# B&R Automation Studio project TD52 (part 55)

### module_EmissionSCR.var - SCR variables
```iecst
VAR
	bAMM_2446 : BOOL := FALSE; (*Warning - SCR BUS communication interrupted [W2446]*) (*V04.05.00.00*)
	bAMM_2447 : BOOL := FALSE; (*Warning - SCR Measuring signal failure urea pressure before dosing [W2447]*) (*V04.05.00.00*)
	bAMM_2448 : BOOL := FALSE; (*Warning - SCR Urea pressure before dosing minimum [W2448]*) (*V04.05.00.00*)
	bAMM_2449 : BOOL := FALSE; (*Warning - SCR Urea pressure before dosing maximum [W2449]*) (*V04.05.00.00*)
	bAMM_2451 : BOOL := FALSE; (*Warning - SCR Urea dosing valve - error [W2451]*) (*V04.05.00.00*)
	bAMM_2452 : BOOL := FALSE; (*Warning - SCR Measuring signal failure urea flow rate after dosing [W2452]*) (*V04.05.00.00*)
	bAMM_2453 : BOOL := FALSE; (*Warning - SCR Urea flow rate - valve characteristic deviating maximum [W2453]*) (*V04.05.00.00*)
	bAMM_2454 : BOOL := FALSE; (*Warning - SCR Compressed air supply pressure urea injection maximum [W2454]*) (*V04.05.00.00*)
	bAMM_2455_CO : BOOL := FALSE; (*Warning - SCR CO Deviation to continous emission monitoring system maximum [W2455]*) (*V04.05.01.00*)
	bAMM_2455_NOx : BOOL := FALSE; (*Warning - SCR NOx Deviation to continous emission monitoring system maximum [W2455]*) (*V04.05.01.00*)
	bAMM_2455_NOxS : BOOL := FALSE; (*Warning - SCR Deviation NOx Sensor to continous emission monitoring system maximum [W2455]*) (*V04.05.01.00*)
	bAMM_2456 : BOOL := FALSE; (*Warning - SCR Emission measurement line 1 - O2 maximum [W2456]*) (*V04.05.00.00*)
	bAMM_2457 : BOOL := FALSE; (*Warning - SCR Measuring signal failure emission measurement line 1 - O2 sensor [W2457]*) (*V04.05.00.00*)
	bAMM_2458 : BOOL := FALSE; (*Warning - SCR Measuring signal failure emission measurement line 2 - NO2 sensor [W2458]*) (*V04.05.00.00*)
	bAMM_2464 : BOOL := FALSE; (*Warning - SCR Urea dosing unit (external) - error [W2464]*) (*V04.05.00.00*)
	bAMM_2697 : BOOL := FALSE; (*Warning - SCR Urea dosing unit - maintenance needed  [W2697]*) (*V04.05.00.00*)
	bAMM_2766 : BOOL := FALSE; (*Warning - Catalyst temperature minimum [W2766]*) (*V04.11.00.00*)
	bAMM_2769 : BOOL := FALSE; (*Warning - SCR Emission measurement air line - moisture maximum [W2769]*) (*V04.14.00.00*)
	bAMM_3379 : BOOL := FALSE; (*Trip - SCR Exhaust temperatures CAT maximum  [A3379]*) (*V04.05.00.00*)
	bAMM_3383 : BOOL := FALSE; (*Trip - SCR Measuring signal failure exhaust temperatures CAT  [A3383]*) (*V04.05.00.00*)
	bAMM_3451 : BOOL := FALSE; (*Warning - SCR Power supply to the valves interrupted [W3451]*) (*V04.05.00.00*)
	bAMM_3452 : BOOL := FALSE; (*Warning - SCR Measuring signal failure urea pressure after dosing [W3452]*) (*V04.05.00.00*)
	bAMM_3453 : BOOL := FALSE; (*Warning - SCR Urea pressure after dosing maximum [W3453]*) (*V04.05.00.00*)
	bAMM_3454 : BOOL := FALSE; (*Warning - SCR Urea pressure after dosing minimum [W3454]*) (*V04.05.00.00*)
	bAMM_3455 : BOOL := FALSE; (*Warning - SCR Urea flow rate after dosing maximum [W3455]*) (*V04.05.00.00*)
	bAMM_3456 : BOOL := FALSE; (*Warning - SCR Urea dosing pump - error [W3456]*) (*V04.05.00.00*)
	bAMM_3457 : BOOL := FALSE; (*Warning - SCR Urea-air valve blocked [W3457]*) (*V04.05.00.00*)
	bAMM_3459 : BOOL := FALSE; (*Warning - SCR Urea tank level minimum - dosing deactivated [W3459]*) (*V04.05.00.00*)
	bAMM_3460 : BOOL := FALSE; (*Warning - SCR Urea supply pump not operating [W3460]*) (*V04.05.00.00*)
	bAMM_3461 : BOOL := FALSE; (*Warning - SCR Measuring signal failure compressed air supply pressure urea injection [W3461]*) (*V04.05.00.00*)
	bAMM_3462 : BOOL := FALSE; (*Warning - SCR Compressed air supply pressure urea injection minimum [W3462]*) (*V04.05.00.00*)
	bAMM_3463 : BOOL := FALSE; (*Warning - SCR Compressed air valve urea injection power supply interrupted [W3463]*) (*V04.05.00.00*)
	bAMM_3464 : BOOL := FALSE; (*Warning - SCR Measuring signal failure exhaust pressure CAT inlet [W3464]*) (*V04.05.00.00*)
	bAMM_3465 : BOOL := FALSE; (*Warning - SCR Measuring signal failure exhaust pressure CAT outlet [W3465]*) (*V04.05.00.00*)
	bAMM_3466 : BOOL := FALSE; (*Warning - SCR Measuring signal failure exhaust temperature CAT inlet [W3466]*) (*V04.05.00.00*)
	bAMM_3467 : BOOL := FALSE; (*Warning - SCR Measuring signal failure exhaust temperature CAT outlet [W3467]*) (*V04.05.00.00*)
	bAMM_3469 : BOOL := FALSE; (*Warning - SCR Exhaust differential pressure CAT maximum [W3469]*) (*V04.05.00.00*)
	bAMM_3470 : BOOL := FALSE; (*Warning - SCR Emission measurement sample gas cooler - error [W3470]*) (*V04.05.00.00*)
	bAMM_3471 : BOOL := FALSE; (*Warning - SCR Emission measurement line 1 - sample gas pump not ready [W3471]*) (*V04.05.00.00*)
	bAMM_3472 : BOOL := FALSE; (*Warning - SCR Emission measurement line 2 - sample gas pump not ready [W3472]*) (*V04.05.00.00*)
	bAMM_3473 : BOOL := FALSE; (*Warning - SCR Emission measurement line 1 - moisture maximum [W3473]*) (*V04.05.00.00*)
	bAMM_3474 : BOOL := FALSE; (*Warning - SCR Emission measurement line 2 - moisture maximum [W3474]*) (*V04.05.00.00*)
	bAMM_3475 : BOOL := FALSE; (*Warning - SCR Emission measurement line 1 - flow rate minimum [W3475]*) (*V04.05.00.00*)
	bAMM_3476 : BOOL := FALSE; (*Warning - SCR Emission measurement line 2 - flow rate minimum [W3476]*) (*V04.05.00.00*)
	bAMM_3477 : BOOL := FALSE; (*Warning - SCR Measuring signal failure emission measurement line 2 - NO sensor [W3477]*) (*V04.05.00.00*)
	bAMM_3478 : BOOL := FALSE; (*Warning - SCR Measuring signal failure emission measurement line 1 - NO sensor [W3478]*) (*V04.05.00.00*)
	bAMM_3479 : BOOL := FALSE; (*Warning - SCR Measuring signal failure emission measurement line 1 - NO2 sensor [W3479]*) (*V04.05.00.00*)
	bAMM_3480 : BOOL := FALSE; (*Warning - SCR NH3 slip detection deactivated  [W3480]*) (*V04.05.00.00*)
	bAMM_3481 : BOOL := FALSE; (*Warning - SCR Measuring signal failure emission measurement line 1 - CO sensor [W3481]*) (*V04.05.00.00*)
	bAMM_3486 : BOOL := FALSE; (*Warning - SCR Urea flow rate after dosing minimum [W3486]*) (*V04.05.00.00*)
	bAMM_3487 : BOOL := FALSE; (*Warning - SCR Exhaust temperature CAT inlet maximum [W3487]*) (*V04.05.00.00*)
	bAMM_3488 : BOOL := FALSE; (*Warning - SCR Exhaust temperature CAT outlet maximum [W3488]*) (*V04.05.00.00*)
	bAMM_9212 : BOOL := FALSE; (*Warning - SCR Air compressor - maintenance needed [W9212]*) (*V04.05.00.00*)
	bAMM_9277 : BOOL := FALSE; (*Warning - SCR Urea dosing stopped - error [W9277]*) (*V04.07.00.00*)
	bAMM_9379 : BOOL := FALSE; (*Warning - SCR Measuring signal failure urea tank level [W9379]*) (*V04.13.00.00*)
	bAMM_9380 : BOOL := FALSE; (*Warning - SCR Urea flow dosing error [W9380]*) (*V04.13.00.00*)
	bEMLine1_Exist : BOOL := FALSE; (*SCR Emission measurement line 1 - exist*) (*V04.13.00.00*)
	bEMLine2_Exist : BOOL := FALSE; (*SCR Emission measurement line 2 - exist*) (*V04.13.00.00*)
	bErr_SCR_BUS : BOOL := FALSE; (*SCR: Bus communication not ok*) (*V04.05.00.00*)
	bOpM_2878 : BOOL := FALSE; (*Operational message - SCR Urea dosing activated  [B2878]*) (*V04.05.00.00*)
	bOpM_2879 : BOOL := FALSE; (*Operational message - SCR Urea dosing deactivated  [B2879]*) (*V04.05.00.00*)
	bOpM_2884 : BOOL := FALSE; (*Operational message - SCR Manual mode on [B2884]*) (*V04.05.00.00*)
	bOpM_2885 : BOOL := FALSE; (*Operational message - SCR Manual mode off [B2885]*) (*V04.05.00.00*)
	bOpM_2923 : BOOL := FALSE; (*Operational message - SCR NH3 slip detection started  [B2923]*) (*V04.05.00.00*)
	bOpM_2924 : BOOL := FALSE; (*Operational message - SCR NH3 slip detection completed  [B2924]*) (*V04.05.00.00*)
	bOpM_9077 : BOOL := FALSE; (*Operational message - SCR NH3 slip detection interrupted  [B9077]*) (*V04.13.00.00*)
	bOpM_9079 : BOOL := FALSE; (*Operational message - SCR Urea dosing - dosing conditions reached [B9079]*) (*V04.13.00.00*)
	bOpM_9080 : BOOL := FALSE; (*Operational message - SCR Urea dosing - dosing conditions ended [B9080]*) (*V04.13.00.00*)
	bOpM_9081 : BOOL := FALSE; (*Operational message - SCR Urea dosing - requested [B9081]*) (*V04.13.00.00*)
	bOpM_9082 : BOOL := FALSE; (*Operational message - SCR Urea dosing - unrequested [B9082]*) (*V04.13.00.00*)
	bRelMon_Lev_UreaTank : BOOL := FALSE; (*release monitoring - urea tank level measuring *) (*V04.13.00.00*)
	bRelMon_T_CatIn : BOOL := FALSE; (*release monitoring - temperature before catalyst*) (*V04.05.00.00*)
	bRelMon_T_CatOut : BOOL := FALSE; (*release monitoring - temperature after catalyst*) (*V04.05.00.00*)
	bRel_Dosing : BOOL := FALSE; (*release dosing*) (*V04.05.00.00*)
	bRel_SCR_UDC : BOOL := FALSE; (*SCR Release urea dosing controller (UDC)*) (*V04.05.00.00*)
	bSCR_DosingLimReached : BOOL := FALSE; (*SCR Limits for dosing release reached*) (*V04.07.00.00*)
END_VAR
VAR CONSTANT
	MODBUS_RTU_MASTER_MAX_ARRAY : UINT := 400; (*Max data (INT) to send/receive *) (*V04.05.00.00*)
END_VAR
VAR
	tInternFlow_SCR_UreaDosingOut : HALioAi_Type; (*SCR Urea flow rate after dosing unit [l/h] (INTERNAL)*) (*V04.05.00.00*)
	tInternPr_SCR_ComprAirSupply : HALioAi_Type; (*SCR Compressed air supply pressure urea injection [bar] (INTERNAL)*) (*V04.05.00.00*)
	tInternPr_SCR_UreaDosingIn : HALioAi_Type; (*SCR Urea pressure before dosing unit [bar] (INTERNAL)*) (*V04.05.00.00*)
	tInternPr_SCR_UreaDosingOut : HALioAi_Type; (*SCR Urea pressure after dosing unit [bar] (INTERNAL)*) (*V04.05.00.00*)
	tInternSCR_InjectValve_Air : HALioDi_Type; (*SCR Urea/Air injection valve - air opened (INTERNAL)*) (*V04.05.00.00*)
	tInternSCR_InjectValve_Urea : HALioDi_Type; (*SCR Urea/Air injection valve - urea opened (INTERNAL)*) (*V04.05.00.00*)
	xTON_bRel_SCR_UDC_5m : TON := (0); (*FuB*)
	xUDC : fUDC := (0); (*FuB*) (*V04.05.00.00*)
END_VAR
```

### Program Logical/Emission/GeneralEM (IEC, version 4.14.0) - general functions

#### GeneralEMCyclic.st
```iecst
(*******************************************************************************
GeneralEM		general functions

This code is confidential and proprietary to the INNIO Company.
It may not be used in any form, or reproduced in any manner,
without the express written permission of the INNIO Company.
Copyright, INNIO Company, 2019

Customized modifications: -
------------------------

History:
-------
V04.05.00.00	22.05.2017	Tinello		new
V04.05.06.00	16.07.2018	Tinello 	Bugfix start speed, bu
V04.07.00.00	11.04.2019	Tinello 	engine motortype included
V04.14.00.00	18.11.2024	Farre		added NOx sensor selection: standard or Low (2023-183)

Instructions for use:
--------------------
Outstandings:
------------
*******************************************************************************)
PROGRAM _CYCLIC

	(* Release Module if ParaSetupOk = TRUE *)
	xTON_ParaSetupOk(IN		:= IN_EM.tPB2MM.bParaSetupOk, PT:= T#10s);
	bRelModul_ParaSetupOk	:= xTON_ParaSetupOk.Q;

	(* operation mode *)
	xOpMode.in	:=	IN_EM.iSt_OpMode;
	xOpMode();

	(* Operation mode selector switch *) 	(* 1= manual; 2= auto; 3= test mode *)
	xTOF_OMSS_MAT(IN	:= (IN_EM.iIdx_OMSS = 1) OR (IN_EM.iIdx_OMSS = 2) OR (IN_EM.iIdx_OMSS = 3), PT := T#10m);
	bOMSS_MAT			:= xTOF_OMSS_MAT.IN;
	bOMSS_MAT_TOF_10m	:= xTOF_OMSS_MAT.Q;

	(* engine start speed reached *)
	xGR_MAXR_StartSpd(In:= IN_EM.rN_EngAct,   Gw := Para.rN_EngStart_LimHi, Hy := Para.rN_EngStart_HyHi);
	xTOF_StartSpd(IN 	:= xGR_MAXR_StartSpd.Q AND bRelModul_ParaSetupOk, 	PT := T#10s);
	xTON_StartSpd_5m(IN := xGR_MAXR_StartSpd.Q AND bRelModul_ParaSetupOk, 	PT := T#5m);

	bStartSpd			:= xTOF_StartSpd.Q;
	bStartSpd_5m		:= xTON_StartSpd_5m.Q;

	(* Engine motortype *)
	xEngType.Motortype 	:= INT_TO_UINT(Para.iEng_Motortype);
	xEngType();

	(* Type of device installed after catalyst *)
	bNOxS_CatOut_Std 	:= Para.iNOxS_CatOut_Device_Type = 0;				(* 0: Standard NOx sensor *)
	bNOxS_CatOut_Low 	:= Para.iNOxS_CatOut_Device_Type = 1;				(* 1: Low NOx sensor *)

END_PROGRAM
```

#### GeneralEM.var
```iecst
VAR
	xGR_MAXR_StartSpd : GR_MAXR := (0); (*Engine start speed passed*)
	xTOF_OMSS_MAT : TOF := (0); (*FuB*)
	xTOF_StartSpd : TOF := (0); (*FuB*)
	xTON_ParaSetupOk : TON := (0); (*FuB*)
	xTON_StartSpd_5m : TON := (0); (*FuB*)
END_VAR
```

### Program Logical/Emission/DefaultEM (IEC, version 4.07.0) - Settings default values

#### DefaultEMCyclic.st
```iecst
(*******************************************************************************
DefaultEM		value set

This code is confidential and proprietary to the INNIO Company.
It may not be used in any form, or reproduced in any manner,
without the express written permission of the INNIO Company.
Copyright, INNIO Company, 2019

Customized modifications: -
------------------------

History:
-------
V4.05.0	05.04.2017	Tinello		new
V4.07.0	23.01.2019	Tinello		add Customer DI's

Instructions for use:
--------------------
Outstandings:
------------
*******************************************************************************)
PROGRAM _CYCLIC

	(* SCR *)
	IN_EM.tFS_SCR_EMLine1_Lo.Di				:= IN_EM.tFS_SCR_EMLine1_Lo.Di				OR NOT IN_EM.tFS_SCR_EMLine1_Lo.GoodQual;
	IN_EM.tFS_SCR_EMLine2_Lo.Di				:= IN_EM.tFS_SCR_EMLine2_Lo.Di				OR NOT IN_EM.tFS_SCR_EMLine2_Lo.GoodQual;
	IN_EM.tLev_SCR_UreaDosingCabinet_Hi.Di	:= IN_EM.tLev_SCR_UreaDosingCabinet_Hi.Di	OR NOT IN_EM.tLev_SCR_UreaDosingCabinet_Hi.GoodQual;
	IN_EM.tLev_SCR_UreaTank_Lo.Di			:= IN_EM.tLev_SCR_UreaTank_Lo.Di			OR NOT IN_EM.tLev_SCR_UreaTank_Lo.GoodQual;
	IN_EM.tSCR_AirCompressor_Rdy.Di			:= IN_EM.tSCR_AirCompressor_Rdy.Di			OR NOT IN_EM.tSCR_AirCompressor_Rdy.GoodQual;
	IN_EM.tSCR_ComprAirValve_Rdy.Di			:= IN_EM.tSCR_ComprAirValve_Rdy.Di			OR NOT IN_EM.tSCR_ComprAirValve_Rdy.GoodQual;
	IN_EM.tSCR_EMCooler_Rdy.Di				:= IN_EM.tSCR_EMCooler_Rdy.Di				OR NOT IN_EM.tSCR_EMCooler_Rdy.GoodQual;
	IN_EM.tSCR_EMPump1_Rdy.Di				:= IN_EM.tSCR_EMPump1_Rdy.Di				OR NOT IN_EM.tSCR_EMPump1_Rdy.GoodQual;
	IN_EM.tSCR_EMPump2_Rdy.Di				:= IN_EM.tSCR_EMPump2_Rdy.Di				OR NOT IN_EM.tSCR_EMPump2_Rdy.GoodQual;
	IN_EM.tSCR_UreaDosingPump_Rdy.Di		:= IN_EM.tSCR_UreaDosingPump_Rdy.Di			OR NOT IN_EM.tSCR_UreaDosingPump_Rdy.GoodQual;
	IN_EM.tSCR_UreaDosingPump2_Rdy.Di		:= IN_EM.tSCR_UreaDosingPump2_Rdy.Di		OR NOT IN_EM.tSCR_UreaDosingPump2_Rdy.GoodQual;
	IN_EM.tSCR_UreaSupplyPump_Op.Di			:= IN_EM.tSCR_UreaSupplyPump_Op.Di			OR NOT IN_EM.tSCR_UreaSupplyPump_Op.GoodQual;
	IN_EM.tSCR_ValvePowerSupply_Ok.Di		:= IN_EM.tSCR_ValvePowerSupply_Ok.Di		OR NOT IN_EM.tSCR_ValvePowerSupply_Ok.GoodQual;
	IN_EM.tSCR_InjectValve_Opened.Di		:= IN_EM.tSCR_InjectValve_Opened.Di			OR NOT IN_EM.tSCR_InjectValve_Opened.GoodQual;
	IN_EM.tSCR_Catalyst_Rdy.Di				:= IN_EM.tSCR_Catalyst_Rdy.Di				OR NOT IN_EM.tSCR_Catalyst_Rdy.GoodQual;
	IN_EM.tT_SCR_Cat_HiHi.Di				:= IN_EM.tT_SCR_Cat_HiHi.Di					OR NOT IN_EM.tT_SCR_Cat_HiHi.GoodQual;
END_PROGRAM
```

### Program Logical/Emission/EmissionMon (IEC, version 4.11.0) - + Emission Monitoring 

- EmissionMon.st (not readable text: treated as protected, skipped)

#### EmissionMon.var - Local variables
```iecst
VAR
	bAMM_NOx_Em_AvgDaily_Hi_Ack : BOOL := FALSE; (*NOx emissions - daily average high warning - acknowledgeable*)
	bNewDay : BOOL := FALSE; (*day changed*)
	bNOxValue_Valid : BOOL := FALSE; (*Valid NOx value available*)
	bNOx_Em_EngOut_mg_LoadSet_Save : BOOL := FALSE; (*SAVE Parameter value: NOx emissions at the engine outlet - Load dependent setpoint enable*)
	bP_Act_Min_reached : BOOL := FALSE; (*Minimal power reached*)
	bRelMon_NOx_Em_Avg : BOOL := FALSE; (*Release monitoring of NOx average*)
	i : INT := 0; (*auxiliary variable*)
	iCnt_Em_AvgShort : UINT := 0; (*counter - for average calculation - NOx and CO short-term*)
	iCnt_MonLim_Exc : UINT; (*counter for emission tolerance exceedance [s]*)
	rCO_Em_AvgShort_Sum_mg : REAL := 0; (*Sum for average calculation - CO short-term [mg/Nm3]*)
	rCO_Em_Avg_mg : ARRAY[0..1799] OF REAL := [1800(0)]; (*Up to 1800 values (300min) for average calculation of CO [mg/Nm3]*)
	rCO_Em_CatOut_mg : REAL := 0; (*Actual CO value at catalyst outlet [mg/Nm3]*)
	rNO2_Em_CatOut_mg : REAL := 0; (*Actual NO2 value at catalyst outlet [mg/Nm3]*)
	rNOx_Em_AvgShort_Sum_mg : REAL := 0; (*Sum for average calculation - NOx short-term [mg/Nm3]*)
	rNOx_Em_Avg_mg : ARRAY[0..1799] OF REAL := [1800(0)]; (*Up to 1800 values (300min) for average calculation of NOx [mg/Nm3]*)
	rNOx_Em_EngOut_mg_Set_Int : REAL := 0; (*INTERNAL: NOx emissions at engine outlet - setpoint [mg/Nm3]*)
	rNOx_NOxS_CatOut_mg : REAL := 0; (*Actual NOx value at catalyst outlet from NOx sensor [mg/Nm3]*)
	rNO_Em_CatOut_mg : REAL := 0; (*Actual NO value at catalyst outlet [mg/Nm3]*)
	rP_Set_Min_NormHy : REAL := 0; (*Minimal power setpoint related to rP_nom -  hysteresis*)
	tRealTime : rtctime_typ; (*actual time of controller*)
	tRefPoint_NOx_mg_Set : ARRAY[0..3] OF lcrCurveByPoints_TabEntry_type; (*kW/NOx Points for interpolation of NOx emissions at engine outlet - setpoint [mg/Nm3]*)
	xDTGetTime_RPS : DTGetTime; (*getting time of the controller*)
	xFILTER_R_NOx_mg_Set : FILTER_R := (0); (*FuB*)
	xFILTER_R_O2_EngOut_Avg : FILTER_R := (0); (*FuB*)
	xLCRCurveByPoints_NOx_mg_Set : LCRCurveByPoints := (0); (*FuB*)
	xLCRMovAvgFlt_CO_short : LCRMovAvgFlt := (0); (*FuB*)
	xLCRMovAvgFlt_NOx_daily : LCRMovAvgFlt := (0); (*FuB*)
	xLCRMovAvgFlt_NOx_dailyT : LCRMovAvgFlt := (0); (*FuB*)
	xLCRMovAvgFlt_NOx_short : LCRMovAvgFlt := (0); (*FuB*)
	xTON_10sec_Tick : TON := (0); (*FuB*)
	xTON_CO_Hi_1 : TON := (0); (*FuB*)
	xTON_DosExt_3m : TON := (0); (*FuB*)
	xTON_EngineSteadyState : TON := (0); (*FuB*)
	xTON_GasAnalys_Done : TON := (0); (*FuB*)
	xTON_NOx_Hi_1 : TON := (0); (*FuB*)
	xTON_NOx_Hi_2 : TON := (0); (*FuB*)
	xTON_P_Act_MinHy : TON := (0); (*FuB*)
	xTON_P_Min_02m : TON := (0); (*FuB*)
	xTON_P_Min_20m : TON := (0); (*FuB*)
	xTON_SecondTick : TON := (0); (*FuB*)
	xTON_StartupDone : TON := (0); (*FuB*)
	xTP_30s : TP; (*FuB*)
END_VAR
```

### Program Logical/Emission/NOxSensor (IEC, version 4.14.0) - + Read Nox Data

- NOxSensor.st (not readable text: treated as protected, skipped)

#### NOxSensor.var - Local variables
```iecst
VAR
	bAMM_NOxS_CANrd_CatOut : BOOL := FALSE; (*Warning: No connection to the sensor - NOx sensor CAT out*) (*OldName: newPV; Cycle: 5*)
	bAMM_NOxS_CANrd_EngOut : BOOL := FALSE; (*Warning: No connection to the sensor - NOx sensor engine out*) (*OldName: newPV; Cycle: 5*)
	bAMM_NOxS_CANrd_EngOut_A : BOOL := FALSE; (*Warning: No connection to the sensor - NOx sensor engine out bank A*) (*OldName: newPV; Cycle: 5*)
	bAMM_NOxS_CANrd_EngOut_B : BOOL := FALSE; (*Warning: No connection to the sensor - NOx sensor engine out bank B*) (*OldName: newPV; Cycle: 5*)
	bDewpoint_NOxS1_IF1 : BOOL := FALSE; (*NOx sensors 1 at CAN interface 1 - Dewpoint reached/sensor started*) (*OldName: newPV; Cycle: 5*)
	bDewpoint_NOxS2_IF1 : BOOL := FALSE; (*NOx sensors 2 at CAN interface 1 - Dewpoint reached/sensor started*) (*OldName: newPV; Cycle: 5*)
	bDewpoint_NOxS2_IF2 : BOOL := FALSE; (*NOx sensors 2 at CAN interface 2 - Dewpoint reached/sensor started*) (*OldName: newPV; Cycle: 5*)
	bDewP_Reached_CatOut : BOOL := FALSE; (*Dew point reached - CAT out*) (*OldName: newPV; Cycle: 5*)
	bDewP_Reached_EngOut : BOOL := FALSE; (*Dew point reached - engine out*) (*OldName: newPV; Cycle: 5*)
	bNOxS_CatOut_Diag_Req : BOOL := FALSE; (*NOx sensor - CAT out- self diagnosis request*) (*OldName: newPV; Cycle: 5*)
	bNOxS_CatOut_Diag_Active : BOOL := FALSE; (*NOx sensor - CAT out - self diagnosis active*) (*OldName: newPV; Cycle: 5*)
	bNOxS_EngOut_A_Diag_Active : BOOL := FALSE; (*NOx sensor - engine out bank A - self diagnosis active*) (*OldName: newPV; Cycle: 5*)
	bNOxS_EngOut_A_Diag_Req : BOOL := FALSE; (*NOx sensor - engine out bank A - self diagnosis request *) (*OldName: newPV; Cycle: 5*)
	bNOxS_EngOut_B_Diag_Active : BOOL := FALSE; (*NOx sensor - engine out bank B - self diagnosis active*) (*OldName: newPV; Cycle: 5*)
	bNOxS_EngOut_B_Diag_Req : BOOL := FALSE; (*NOx sensor - engine out bank B - self diagnosis request *) (*OldName: newPV; Cycle: 5*)
	bNOxS_EngOut_Diag_Active : BOOL := FALSE; (*NOx sensor - engine out - self diagnosis active*) (*OldName: newPV; Cycle: 5*)
	bNOxS_EngOut_Diag_Req : BOOL := FALSE; (*NOx sensor - engine out - self diagnosis request *) (*OldName: newPV; Cycle: 5*)
	bQueue_NOxS1_IF1_Done : BOOL := FALSE; (*initialisation of CAN queue for NOx sensor 1 (interface1) is done*) (*OldName: newPV; Cycle: 5*)
	bQueue_NOxS2_IF1_Done : BOOL := FALSE; (*initialisation of CAN queue for NOx sensor 2 (interface1) is done*) (*OldName: newPV; Cycle: 5*)
	bQueue_NOxS2_IF2_Done : BOOL := FALSE; (*initialisation of CAN queue for NOx sensor 2 (interface2) is done*) (*OldName: newPV; Cycle: 5*)
	bRelMon_O2_NOxS_CatOut : BOOL := FALSE; (*Release monitoring NOx sensor at CAT outlet - O2 value*) (*OldName: newPV; Cycle: 5*)
	bRelMon_O2_NOxS_EngOut : BOOL := FALSE; (*Release monitoring NOx sensor at engine outlet - O2 value*) (*OldName: newPV; Cycle: 5*)
	bRelMon_O2_NOxS_EngOut_A : BOOL := FALSE; (*Release monitoring NOx sensor at engine outlet bank A - O2 value*) (*OldName: newPV; Cycle: 5*)
	bRelMon_O2_NOxS_EngOut_B : BOOL := FALSE; (*Release monitoring NOx sensor at engine outlet bank B - O2 value*) (*OldName: newPV; Cycle: 5*)
	bReq_NOxS1_IF1_CF : BOOL := FALSE; (*request correction factor for NOx sensor 1 (interface1)*) (*OldName: newPV; Cycle: 5*)
	bReq_NOxS1_IF1_DiagRes : BOOL := FALSE; (*request self diagnosis result value for NOx sensor 1 (interface1)*) (*OldName: newPV; Cycle: 5*)
	bReq_NOxS1_IF1_OpH : BOOL := FALSE; (*request operating hours for NOx sensor 1 (interface1)*) (*OldName: newPV; Cycle: 5*)
	bReq_NOxS2_IF1_CF : BOOL := FALSE; (*request correction factor for NOx sensor 2 (interface1)*) (*OldName: newPV; Cycle: 5*)
	bReq_NOxS2_IF1_DiagRes : BOOL := FALSE; (*request self diagnosis result value for NOx sensor 2 (interface1)*) (*OldName: newPV; Cycle: 5*)
	bReq_NOxS2_IF1_OpH : BOOL := FALSE; (*request operating hours for NOx sensor 2 (interface1)*) (*OldName: newPV; Cycle: 5*)
	bReq_NOxS2_IF2_CF : BOOL := FALSE; (*request correction factor for NOx sensor 2 (interface2)*) (*OldName: newPV; Cycle: 5*)
	bReq_NOxS2_IF2_DiagRes : BOOL := FALSE; (*request self diagnosis result value for NOx sensor 2 (interface2)*) (*OldName: newPV; Cycle: 5*)
	bReq_NOxS2_IF2_OpH : BOOL := FALSE; (*request operating hours for NOx sensor 2 (interface2)*) (*OldName: newPV; Cycle: 5*)
	bStart_NOxS_CatOut : BOOL := FALSE; (*NOx sensor - CAT out - start command*) (*OldName: newPV; Cycle: 5*)
	bStart_NOxS_EngOut : BOOL := FALSE; (*NOx sensor - engine out - start command*) (*OldName: newPV; Cycle: 5*)
	DATA_NOxS_R : ARRAY[0..7] OF USINT; (*read data from NOx sensor*) (*OldName: newPV; Cycle: 5*)
	DATA_NOxS_W : ARRAY[0..2] OF USINT; (*request data from NOx sensor*) (*OldName: newPV; Cycle: 5*)
	i : UINT := 0; (*auxiliaries variable*) (*OldName: newPV; Cycle: 5*)
	iAlternate_Req : USINT := 0; (*Alternate request*) (*OldName: newPV; Cycle: 5*)
	iCANqueue_NOxS_size : UINT := 0; (*CANqueue size*) (*OldName: newPV; Cycle: 5*)
	iCANwrite_NOxS_Diag_IF1 : ARRAY[0..7] OF USINT; (*Message for NOx sensors CAN interface 1 - self diagnosis*) (*OldName: newPV; Cycle: 5*)
	iCANwrite_NOxS_Diag_IF2 : ARRAY[0..7] OF USINT; (*Message for NOx sensors CAN interface 2 - self diagnosis*) (*OldName: newPV; Cycle: 5*)
	iCANwrite_NOxS_IF1 : ARRAY[0..7] OF USINT; (*Message for NOx sensors CAN interface 1*) (*OldName: newPV; Cycle: 5*)
	iCANwrite_NOxS_IF1_Old : USINT := 0; (*Message for NOx sensors CAN interface 1 - saved*) (*OldName: newPV; Cycle: 5*)
	iCANwrite_NOxS_IF2 : ARRAY[0..7] OF USINT; (*Message for NOx sensors CAN interface 2*) (*OldName: newPV; Cycle: 5*)
	iCANwrite_NOxS_IF2_Old : USINT := 0; (*Message for NOx sensors CAN interface 2 - saved*) (*OldName: newPV; Cycle: 5*)
	iCAN_NOxS_us_ident : UDINT; (*identifier for CAN read/write*) (*OldName: newPV; Cycle: 5*)
	iCnt_NOxS_CatOut_Diag : USINT := 0; (*Counter - NOx sensor catalyst out - diagnosis counter*) (*OldName: newPV; Cycle: 5*)
	iCnt_NOxS_EngOut_A_Diag : USINT := 0; (*Counter - NOx sensor engine out A - diagnosis counter*) (*OldName: newPV; Cycle: 5*)
	iCnt_NOxS_EngOut_B_Diag : USINT := 0; (*Counter - NOx sensor engine out B - diagnosis counter*) (*OldName: newPV; Cycle: 5*)
	iCnt_NOxS_EngOut_Diag : USINT := 0; (*Counter - NOx sensor engine out - diagnosis counter*) (*OldName: newPV; Cycle: 5*)
	iCnt_NOx_NOxS_CatOut_Err : USINT := 0; (*Counter - NOx sensor catalyst out - error NOx*) (*OldName: newPV; Cycle: 5*)
	iCnt_NOx_NOxS_EngOut_A_Err : USINT := 0; (*Counter - NOx sensor engine out A - error NOx*) (*OldName: newPV; Cycle: 5*)
	iCnt_NOx_NOxS_EngOut_B_Err : USINT := 0; (*Counter - NOx sensor engine out B - error NOx*) (*OldName: newPV; Cycle: 5*)
	iCnt_NOx_NOxS_EngOut_Err : USINT := 0; (*Counter - NOx sensor engine out - error NOx*) (*OldName: newPV; Cycle: 5*)
	iCnt_O2_NOxS_CatOut_Err : USINT := 0; (*Counter - NOx sensor catalyst out - error O2*) (*OldName: newPV; Cycle: 5*)
	iCnt_O2_NOxS_EngOut_A_Err : USINT := 0; (*Counter - NOx sensor engine out A - error O2*) (*OldName: newPV; Cycle: 5*)
	iCnt_O2_NOxS_EngOut_B_Err : USINT := 0; (*Counter - NOx sensor engine out B - error O2*) (*OldName: newPV; Cycle: 5*)
	iCnt_O2_NOxS_EngOut_Err : USINT := 0; (*Counter - NOx sensor engine out - error O2*) (*OldName: newPV; Cycle: 5*)
	iCnt_OpHours_Old : DINT; (*Save operating hours*) (*OldName: newPV; Cycle: 5*)
	iCnt_RequestTrials : ARRAY[0..9] OF USINT; (*Number of request trials*) (*OldName: newPV; Cycle: 5*)
	iCnt_Wait : USINT := 0; (*Cycle counter - wait for CAN message*) (*OldName: newPV; Cycle: 5*)
	iCnt_WaitErrS1_IF1 : USINT := 0; (*Cycle counter - error while waiting for CAN message*) (*OldName: newPV; Cycle: 5*)
	iCnt_WaitErrS2_IF1 : USINT := 0; (*Cycle counter - error while waiting for CAN message*) (*OldName: newPV; Cycle: 5*)
	iCnt_WaitErrS2_IF2 : USINT := 0; (*Cycle counter - error while waiting for CAN message*) (*OldName: newPV; Cycle: 5*)
	iCnt_WaitS1_IF1 : USINT := 0; (*Cycle counter - wait for CAN message*) (*OldName: newPV; Cycle: 5*)
	iCnt_WaitS2_IF1 : USINT := 0; (*Cycle counter - wait for CAN message*) (*OldName: newPV; Cycle: 5*)
	iCnt_WaitS2_IF2 : USINT := 0; (*Cycle counter - wait for CAN message*) (*OldName: newPV; Cycle: 5*)
	iIdx_NOxS_Config_Old : INT := 0; (*Save - PARA: NOx  Sensor configuration*) (*OldName: newPV; Cycle: 5*)
	iNOx_NOxS_CatOut_Wet : UINT := 0; (*NOx sensor catalyst out - assembly high and low byte of NOx*) (*OldName: newPV; Cycle: 5*)
	iNOx_NOxS_EngOut_A_Wet : UINT := 0; (*NOx sensor engine out A - assembly high and low byte of NOx*) (*OldName: newPV; Cycle: 5*)
	iNOx_NOxS_EngOut_B_Wet : UINT := 0; (*NOx sensor engine out B - assembly high and low byte of NOx*) (*OldName: newPV; Cycle: 5*)
	iNOx_NOxS_EngOut_Wet : UINT := 0; (*NOx sensor engine out - assembly high and low byte of NOx*) (*OldName: newPV; Cycle: 5*)
	iO2_NOxS_CatOut_Wet : UINT := 0; (*NOx sensor catalyst out - assembly high and low byte of O2*) (*OldName: newPV; Cycle: 5*)
	iO2_NOxS_EngOut_A_Wet : UINT := 0; (*NOx sensor engine out A - assembly high and low byte of O2*) (*OldName: newPV; Cycle: 5*)
	iO2_NOxS_EngOut_B_Wet : UINT := 0; (*NOx sensor engine out B - assembly high and low byte of O2*) (*OldName: newPV; Cycle: 5*)
	iO2_NOxS_EngOut_Wet : UINT := 0; (*NOx sensor engine out - assembly high and low byte of O2*) (*OldName: newPV; Cycle: 5*)
	iRead_NOxS_CatOut : ARRAY[0..7] OF USINT; (*CAN data - NOx sensor catalyst out*) (*OldName: newPV; Cycle: 5*)
	iRead_NOxS_EngOut : ARRAY[0..7] OF USINT; (*CAN data - NOx sensor engine out*) (*OldName: newPV; Cycle: 5*)
	iRead_NOxS_EngOut_A : ARRAY[0..7] OF USINT; (*CAN data - NOx sensor engine out A*) (*OldName: newPV; Cycle: 5*)
	iRead_NOxS_EngOut_B : ARRAY[0..7] OF USINT; (*CAN data - NOx sensor engine out B*) (*OldName: newPV; Cycle: 5*)
	iSel_NOxS_Request : USINT := 0; (*Selection of CAN request*) (*OldName: newPV; Cycle: 5*)
	iSt_NOxS_CatOut_Diagnosis : USINT := 0; (*NOx sensor catalyst out - status diagnosis feedback*) (*OldName: newPV; Cycle: 5*)
	iSt_NOxS_CatOut_HeaterErr : USINT := 0; (*NOx sensor catalyst out - status heater error*) (*OldName: newPV; Cycle: 5*)
	iSt_NOxS_CatOut_HeaterMode : USINT := 0; (*NOx sensor catalyst out - status heater mode*) (*OldName: newPV; Cycle: 5*)
	iSt_NOxS_CatOut_HeaterTemp : USINT := 0; (*NOx sensor catalyst out - status temperature heater*) (*OldName: newPV; Cycle: 5*)
	iSt_NOxS_CatOut_NOxErr : USINT := 0; (*NOx sensor catalyst out - status NOx error*) (*OldName: newPV; Cycle: 5*)
	iSt_NOxS_CatOut_NOxSignal : USINT := 0; (*NOx sensor catalyst out - status NOx signal*) (*OldName: newPV; Cycle: 5*)
	iSt_NOxS_CatOut_O2Err : USINT := 0; (*NOx sensor catalyst out - status Oxygen error*) (*OldName: newPV; Cycle: 5*)
	iSt_NOxS_CatOut_O2Signal : USINT := 0; (*NOx sensor catalyst out - status Oxygen signal*) (*OldName: newPV; Cycle: 5*)
	iSt_NOxS_CatOut_PowerRange : USINT := 0; (*NOx sensor catalyst out - status power in range*) (*OldName: newPV; Cycle: 5*)
	iSt_NOxS_EngOut_A_Diagnosis : USINT := 0; (*NOx sensor engine out A - status diagnosis feedback*) (*OldName: newPV; Cycle: 5*)
	iSt_NOxS_EngOut_A_HeaterErr : USINT := 0; (*NOx sensor engine out A - status heater error*) (*OldName: newPV; Cycle: 5*)
	iSt_NOxS_EngOut_A_HeaterMode : USINT := 0; (*NOx sensor engine out A - status heater mode*) (*OldName: newPV; Cycle: 5*)
	iSt_NOxS_EngOut_A_HeaterTemp : USINT := 0; (*NOx sensor engine out A - status temperature heater*) (*OldName: newPV; Cycle: 5*)
	iSt_NOxS_EngOut_A_NOxErr : USINT := 0; (*NOx sensor engine out A - status NOx error*) (*OldName: newPV; Cycle: 5*)
	iSt_NOxS_EngOut_A_NOxSignal : USINT := 0; (*NOx sensor engine out A - status NOx signal*) (*OldName: newPV; Cycle: 5*)
	iSt_NOxS_EngOut_A_O2Err : USINT := 0; (*NOx sensor engine out A - status Oxygen error*) (*OldName: newPV; Cycle: 5*)
	iSt_NOxS_EngOut_A_O2Signal : USINT := 0; (*NOx sensor engine out A - status Oxygen signal*) (*OldName: newPV; Cycle: 5*)
	iSt_NOxS_EngOut_A_PowerRange : USINT := 0; (*NOx sensor engine out A - status power in range*) (*OldName: newPV; Cycle: 5*)
	iSt_NOxS_EngOut_B_Diagnosis : USINT := 0; (*NOx sensor engine out B - status diagnosis feedback*) (*OldName: newPV; Cycle: 5*)
	iSt_NOxS_EngOut_B_HeaterErr : USINT := 0; (*NOx sensor engine out B - status heater error*) (*OldName: newPV; Cycle: 5*)
	iSt_NOxS_EngOut_B_HeaterMode : USINT := 0; (*NOx sensor engine out B - status heater mode*) (*OldName: newPV; Cycle: 5*)
	iSt_NOxS_EngOut_B_HeaterTemp : USINT := 0; (*NOx sensor engine out B - status temperature heater*) (*OldName: newPV; Cycle: 5*)
	iSt_NOxS_EngOut_B_NOxErr : USINT := 0; (*NOx sensor engine out B - status NOx error*) (*OldName: newPV; Cycle: 5*)
	iSt_NOxS_EngOut_B_NOxSignal : USINT := 0; (*NOx sensor engine out B - status NOx signal*) (*OldName: newPV; Cycle: 5*)
	iSt_NOxS_EngOut_B_O2Err : USINT := 0; (*NOx sensor engine out B - status Oxygen error*) (*OldName: newPV; Cycle: 5*)
	iSt_NOxS_EngOut_B_O2Signal : USINT := 0; (*NOx sensor engine out B - status Oxygen signal*) (*OldName: newPV; Cycle: 5*)
	iSt_NOxS_EngOut_B_PowerRange : USINT := 0; (*NOx sensor engine out B - status power in range*) (*OldName: newPV; Cycle: 5*)
	iSt_NOxS_EngOut_Diagnosis : USINT := 0; (*NOx sensor engine out - status diagnosis feedback*) (*OldName: newPV; Cycle: 5*)
	iSt_NOxS_EngOut_HeaterErr : USINT := 0; (*NOx sensor engine out - status heater error*) (*OldName: newPV; Cycle: 5*)
	iSt_NOxS_EngOut_HeaterMode : USINT := 0; (*NOx sensor engine out - status heater mode*) (*OldName: newPV; Cycle: 5*)
	iSt_NOxS_EngOut_HeaterTemp : USINT := 0; (*NOx sensor engine out - status temperature heater*) (*OldName: newPV; Cycle: 5*)
	iSt_NOxS_EngOut_NOxErr : USINT := 0; (*NOx sensor engine out - status NOx error*) (*OldName: newPV; Cycle: 5*)
	iSt_NOxS_EngOut_NOxSignal : USINT := 0; (*NOx sensor engine out - status NOx signal*) (*OldName: newPV; Cycle: 5*)
	iSt_NOxS_EngOut_O2Err : USINT := 0; (*NOx sensor engine out - status Oxygen error*) (*OldName: newPV; Cycle: 5*)
	iSt_NOxS_EngOut_O2Signal : USINT := 0; (*NOx sensor engine out - status Oxygen signal*) (*OldName: newPV; Cycle: 5*)
	iSt_NOxS_EngOut_PowerRange : USINT := 0; (*NOx sensor engine out - status power in range*) (*OldName: newPV; Cycle: 5*)
	iSt_ReadOut : USINT := 0; (*State - CAN request*) (*OldName: newPV; Cycle: 5*)
	rCntNOx_NOxS_CatOut_Ok : REAL := 0; (*counter - messages from NOx sensor after catalyst without NOx error*) (*OldName: newPV; Cycle: 5*)
	rCntNOx_NOxS_EngOut_A_Ok : REAL := 0; (*counter - messages from NOx sensor after engine A without NOx error*) (*OldName: newPV; Cycle: 5*)
	rCntNOx_NOxS_EngOut_B_Ok : REAL := 0; (*counter - messages from NOx sensor after engine B without NOx error*) (*OldName: newPV; Cycle: 5*)
	rCntNOx_NOxS_EngOut_Ok : REAL := 0; (*counter - messages from NOx sensor after engine without NOx error*) (*OldName: newPV; Cycle: 5*)
	rCntO2_NOxS_CatOut_Ok : REAL := 0; (*counter - messages from NOx sensor after catalyst without O2 error*) (*OldName: newPV; Cycle: 5*)
	rCntO2_NOxS_EngOut_A_Ok : REAL := 0; (*counter - messages from NOx sensor after engine A without O2 error*) (*OldName: newPV; Cycle: 5*)
	rCntO2_NOxS_EngOut_B_Ok : REAL := 0; (*counter - messages from NOx sensor after engine B without O2 error*) (*OldName: newPV; Cycle: 5*)
	rCntO2_NOxS_EngOut_Ok : REAL := 0; (*counter - messages from NOx sensor after engine without O2 error*) (*OldName: newPV; Cycle: 5*)
	rk_NO2_NOxS_CatOut : REAL := 0.8; (*NOx sensor at catalyst outlet - NO2 cross sensitivity correction factor [%]*) (*OldName: newPV; Cycle: 5*)
	rk_NO2_NOxS_EngOut : REAL := 0.8; (*NOx sensor at engine outlet - NO2 cross sensitivity correction factor [%]*) (*OldName: newPV; Cycle: 5*)
	rk_NO2_NOxS_EngOut_A : REAL := 0.8; (*NOx sensor at engine outlet A - NO2 cross sensitivity correction factor [%]*) (*OldName: newPV; Cycle: 5*)
	rk_NO2_NOxS_EngOut_B : REAL := 0.8; (*NOx sensor at engine outlet B - NO2 cross sensitivity correction factor [%]*) (*OldName: newPV; Cycle: 5*)
	rNOx_NOxS_CatOut_Dry : REAL := 0; (*NOx sensor at catalyst outlet - actual NOx value [ppm]*) (*OldName: newPV; Cycle: 5*)
	rNOx_NOxS_CatOut_DurDiag_P1 : REAL := 0; (*NOx sensor at catalyst outlet - NOx value during self diagnosis [ppm wet]*) (*OldName: newPV; Cycle: 5*)
	rNOx_NOxS_CatOut_Wet : REAL := 0; (*NOx sensor at catalyst outlet - actual NOx value [ppm wet]*) (*OldName: newPV; Cycle: 5*)
	rNOx_NOxS_CatOut_Wet_Cor : REAL := 0; (*NOx sensor at catalyst outlet - actual NOx value corrected by cross sensitivity [ppm wet]*) (*OldName: newPV; Cycle: 5*)
	rNOx_NOxS_CatOut_Wet_Save : REAL := 0; (*NOx sensor at catalyst outlet - actual NOx value - saved [ppm wet]*) (*OldName: newPV; Cycle: 5*)
	rNOx_NOxS_CatOut_Wet_Sum : REAL := 0; (*NOx sensor at catalyst outlet - sum of NOx value from last queue [ppm wet]*) (*OldName: newPV; Cycle: 5*)
	rNOx_NOxS_EngOut_A_Dry : REAL := 0; (*NOx sensor at engine outlet A - actual NOx value [ppm]*) (*OldName: newPV; Cycle: 5*)
	rNOx_NOxS_EngOut_A_DurDiag_P1 : REAL := 0; (*NOx sensor at engine outlet A - NOx value during self diagnosis [ppm wet]*) (*OldName: newPV; Cycle: 5*)
	rNOx_NOxS_EngOut_A_Wet : REAL := 0; (*NOx sensor at engine outlet A - actual NOx value [ppm wet]*) (*OldName: newPV; Cycle: 5*)
	rNOx_NOxS_EngOut_A_Wet_Cor : REAL := 0; (*NOx sensor at engine outlet A - actual NOx value corrected by cross sensitivity [ppm wet]*) (*OldName: newPV; Cycle: 5*)
	rNOx_NOxS_EngOut_A_Wet_Save : REAL := 0; (*NOx sensor at engine outlet A - actual NOx value - saved [ppm wet]*) (*OldName: newPV; Cycle: 5*)
	rNOx_NOxS_EngOut_A_Wet_Sum : REAL := 0; (*NOx sensor at engine outlet A - sum of NOx value from last queue [ppm wet]*) (*OldName: newPV; Cycle: 5*)
	rNOx_NOxS_EngOut_B_Dry : REAL := 0; (*NOx sensor at engine outlet B - actual NOx value [ppm]*) (*OldName: newPV; Cycle: 5*)
	rNOx_NOxS_EngOut_B_DurDiag_P1 : REAL := 0; (*NOx sensor at engine outlet B - NOx value during self diagnosis [ppm wet]*) (*OldName: newPV; Cycle: 5*)
	rNOx_NOxS_EngOut_B_Wet : REAL := 0; (*NOx sensor at engine outlet B - actual NOx value [ppm wet]*) (*OldName: newPV; Cycle: 5*)
	rNOx_NOxS_EngOut_B_Wet_Cor : REAL := 0; (*NOx sensor at engine outlet B - actual NOx value corrected by cross sensitivity [ppm wet]*) (*OldName: newPV; Cycle: 5*)
	rNOx_NOxS_EngOut_B_Wet_Save : REAL := 0; (*NOx sensor at engine outlet B - actual NOx value - saved [ppm wet]*) (*OldName: newPV; Cycle: 5*)
	rNOx_NOxS_EngOut_B_Wet_Sum : REAL := 0; (*NOx sensor at engine outlet B - sum of NOx value from last queue [ppm wet]*) (*OldName: newPV; Cycle: 5*)
	rNOx_NOxS_EngOut_Dry : REAL := 0; (*NOx sensor at engine outlet - actual NOx value [ppm]*) (*OldName: newPV; Cycle: 5*)
	rNOx_NOxS_EngOut_DurDiag_P1 : REAL := 0; (*NOx sensor at engine outlet - NOx value during self diagnosis [ppm wet]*) (*OldName: newPV; Cycle: 5*)
	rNOx_NOxS_EngOut_Wet : REAL := 0; (*NOx sensor at engine outlet - actual NOx value [ppm wet]*) (*OldName: newPV; Cycle: 5*)
	rNOx_NOxS_EngOut_Wet_Cor : REAL := 0; (*NOx sensor at engine outlet - actual NOx value corrected by cross sensitivity [ppm wet]*) (*OldName: newPV; Cycle: 5*)
	rNOx_NOxS_EngOut_Wet_Save : REAL := 0; (*NOx sensor at engine outlet - actual NOx value - saved [ppm wet]*) (*OldName: newPV; Cycle: 5*)
	rNOx_NOxS_EngOut_Wet_Sum : REAL := 0; (*NOx sensor at engine outlet - sum of NOx value from last queue [ppm wet]*) (*OldName: newPV; Cycle: 5*)
	rO2_EngOut : REAL := 0; (*Dry O2 value at engine outlet [Vol%] which is used to transform NOx (ppm -> mg/Nm3 or from mg/Nm3 -> ppm)*) (*OldName: newPV; Cycle: 5*)
	rO2_EngOut_A : REAL := 0; (*Dry O2 value at engine outlet A [Vol%] which is used to transform NOx (ppm -> mg/Nm3 or from mg/Nm3 -> ppm)*) (*OldName: newPV; Cycle: 5*)
	rO2_EngOut_B : REAL := 0; (*Dry O2 value at engine outlet B [Vol%] which is used to transform NOx (ppm -> mg/Nm3 or from mg/Nm3 -> ppm)*) (*OldName: newPV; Cycle: 5*)
	rO2_Lambda_Dry : REAL := 0; (*Calculated dry O2 value out of Lambda [Vol%]*) (*OldName: newPV; Cycle: 5*)
	rO2_Lambda_Wet : REAL := 0; (*Calculated wet O2 value out of Lambda [Vol% wet]*) (*OldName: newPV; Cycle: 5*)
	rO2_NOxS_Avg_Wet_Offs : REAL := 0; (*NOx sensor average - offset corrected wet O2 value out of all active NOx sensors [Vol% wet]*) (*OldName: newPV; Cycle: 5*)
	rO2_NOxS_CatOut_Dry : REAL := 0; (*NOx sensor at catalyst outlet - actual O2 value [Vol%]*) (*OldName: newPV; Cycle: 5*)
	rO2_NOxS_CatOut_DurDiag_P1 : REAL := 0; (*NOx sensor at catalyst outlet - O2 value during self diagnosis [Vol% wet]*) (*OldName: newPV; Cycle: 5*)
	rO2_NOxS_CatOut_Wet : REAL := 0; (*NOx sensor at catalyst outlet - actual O2 value [Vol% wet]*) (*OldName: newPV; Cycle: 5*)
	rO2_NOxS_CatOut_Wet_Save : REAL := 0; (*NOx sensor at catalyst outlet - actual O2 value - saved [Vol% wet]*) (*OldName: newPV; Cycle: 5*)
	rO2_NOxS_CatOut_Wet_Sum : REAL := 0; (*NOx sensor at catalyst outlet - sum of O2 value from last queue [Vol% wet]*) (*OldName: newPV; Cycle: 5*)
	rO2_NOxS_EngOut_A_Dry : REAL := 0; (*NOx sensor at engine outlet A - actual O2 value [Vol%]*) (*OldName: newPV; Cycle: 5*)
	rO2_NOxS_EngOut_A_DurDiag_P1 : REAL := 0; (*NOx sensor at engine outlet A - O2 value during self diagnosis [Vol% wet]*) (*OldName: newPV; Cycle: 5*)
	rO2_NOxS_EngOut_A_Wet : REAL := 0; (*NOx sensor at engine outlet A - actual O2 value [Vol% wet]*) (*OldName: newPV; Cycle: 5*)
	rO2_NOxS_EngOut_A_Wet_Save : REAL := 0; (*NOx sensor at engine outlet A - actual O2 value - saved [Vol% wet]*) (*OldName: newPV; Cycle: 5*)
	rO2_NOxS_EngOut_A_Wet_Sum : REAL := 0; (*NOx sensor at engine outlet A - sum of O2 value from last queue [Vol% wet]*) (*OldName: newPV; Cycle: 5*)
	rO2_NOxS_EngOut_B_Dry : REAL := 0; (*NOx sensor at engine outlet B - actual O2 value [Vol%]*) (*OldName: newPV; Cycle: 5*)
	rO2_NOxS_EngOut_B_DurDiag_P1 : REAL := 0; (*NOx sensor at engine outlet B - O2 value during self diagnosis [Vol% wet]*) (*OldName: newPV; Cycle: 5*)
	rO2_NOxS_EngOut_B_Wet : REAL := 0; (*NOx sensor at engine outlet B - actual O2 value [Vol% wet]*) (*OldName: newPV; Cycle: 5*)
	rO2_NOxS_EngOut_B_Wet_Save : REAL := 0; (*NOx sensor at engine outlet B - actual O2 value - saved [Vol% wet]*) (*OldName: newPV; Cycle: 5*)
	rO2_NOxS_EngOut_B_Wet_Sum : REAL := 0; (*NOx sensor at engine outlet B - sum of O2 value from last queue [Vol% wet]*) (*OldName: newPV; Cycle: 5*)
	rO2_NOxS_EngOut_Dry : REAL := 0; (*NOx sensor at engine outlet - actual O2 value [Vol%]*) (*OldName: newPV; Cycle: 5*)
	rO2_NOxS_EngOut_DurDiag_P1 : REAL := 0; (*NOx sensor at engine outlet - O2 value during self diagnosis [Vol% wet]*) (*OldName: newPV; Cycle: 5*)
	rO2_NOxS_EngOut_Wet : REAL := 0; (*NOx sensor at engine outlet - actual O2 value [Vol% wet]*) (*OldName: newPV; Cycle: 5*)
	rO2_NOxS_EngOut_Wet_Save : REAL := 0; (*NOx sensor at engine outlet - actual O2 value - saved [Vol% wet]*) (*OldName: newPV; Cycle: 5*)
	rO2_NOxS_EngOut_Wet_Sum : REAL := 0; (*NOx sensor at engine outlet - sum of O2 value from last queue [Vol% wet]*) (*OldName: newPV; Cycle: 5*)
	rPc_NOxS_CatOut_DiagResult_Sum : REAL := 0.0; (*NOx sensor catalyst out - sum of diagnosis result*) (*OldName: newPV; Cycle: 5*)
	rPc_NOxS_EngOut_A_DiagResult_Sum : REAL := 0.0; (*NOx sensor engine out A - sum of diagnosis result*) (*OldName: newPV; Cycle: 5*)
	rPc_NOxS_EngOut_B_DiagResult_Sum : REAL := 0.0; (*NOx sensor engine out B - sum of diagnosis result*) (*OldName: newPV; Cycle: 5*)
	rPc_NOxS_EngOut_DiagResult_Sum : REAL := 0.0; (*NOx sensor engine out - sum of diagnosis result*) (*OldName: newPV; Cycle: 5*)
	ti_DewP_CatOut_Add : TIME := 0; (*Additional time until dew point reached in case of missing sensor [s]*) (*OldName: newPV; Cycle: 5*)
	xCANqueue_NOxS1_IF1 : CANqueue := (0); (*FuB*) (*OldName: newPV; Cycle: 5*)
	xCANqueue_NOxS2_IF1 : CANqueue := (0); (*FuB*) (*OldName: newPV; Cycle: 5*)
	xCANqueue_NOxS2_IF2 : CANqueue := (0); (*FuB*) (*OldName: newPV; Cycle: 5*)
	xCANqueue_NOxS2_IF3 : CANqueue := (0); (*FuB*) (*OldName: newPV; Cycle: 5*)
	xCANrd_NOxS_CatOut : CANrd := (0); (*FuB*) (*OldName: newPV; Cycle: 5*)
	xCANrd_NOxS_EngOut : CANrd := (0); (*FuB*) (*OldName: newPV; Cycle: 5*)
	xCANrd_NOxS_EngOut_A : CANrd := (0); (*FuB*) (*OldName: newPV; Cycle: 5*)
	xCANrd_NOxS_EngOut_B : CANrd := (0); (*FuB*) (*OldName: newPV; Cycle: 5*)
	xCANread_NOxS : CANread := (0); (*FuB*) (*OldName: newPV; Cycle: 5*)
	xCANwrite_NOxS : CANwrite := (0); (*FuB*) (*OldName: newPV; Cycle: 5*)
	xCANwrite_NOxS_IF1_DewP : CANwrite := (0); (*FuB*) (*OldName: newPV; Cycle: 5*)
	xCANwrite_NOxS_IF1_Diag : CANwrite := (0); (*FuB*) (*OldName: newPV; Cycle: 5*)
	xCANwrite_NOxS_IF2_DewP : CANwrite := (0); (*FuB*) (*OldName: newPV; Cycle: 5*)
	xCANwrite_NOxS_IF2_Diag : CANwrite := (0); (*FuB*) (*OldName: newPV; Cycle: 5*)
	xFILTER_R_Hum_CatOut : FILTER_R := (0); (*FuB*) (*OldName: newPV; Cycle: 5*)
	xFILTER_R_NOx_NOxS_CatOut : FILTER_R := (0); (*FuB*) (*OldName: newPV; Cycle: 5*)
	xFILTER_R_NOx_NOxS_CatOut_mg : FILTER_R := (0); (*FuB*) (*OldName: newPV; Cycle: 5*)
	xFILTER_R_NOx_NOxS_EngOut : FILTER_R := (0); (*FuB*) (*OldName: newPV; Cycle: 5*)
	xFILTER_R_NOx_NOxS_EngOut_A : FILTER_R := (0); (*FuB*) (*OldName: newPV; Cycle: 5*)
	xFILTER_R_NOx_NOxS_EngOut_Avg : FILTER_R := (0); (*FuB*) (*OldName: newPV; Cycle: 5*)
	xFILTER_R_NOx_NOxS_EngOut_A_mg : FILTER_R := (0); (*FuB*) (*OldName: newPV; Cycle: 5*)
	xFILTER_R_NOx_NOxS_EngOut_B : FILTER_R := (0); (*FuB*) (*OldName: newPV; Cycle: 5*)
	xFILTER_R_NOx_NOxS_EngOut_B_mg : FILTER_R := (0); (*FuB*) (*OldName: newPV; Cycle: 5*)
	xFILTER_R_NOx_NOxS_EngOut_mg : FILTER_R := (0); (*FuB*) (*OldName: newPV; Cycle: 5*)
	xFILTER_R_NOx_NOxS_EngOut_mg_Avg : FILTER_R := (0); (*FuB*) (*OldName: newPV; Cycle: 5*)
	xFILTER_R_O2_NOxS_CatOut : FILTER_R := (0); (*FuB*) (*OldName: newPV; Cycle: 5*)
	xFILTER_R_O2_NOxS_EngOut : FILTER_R := (0); (*FuB*) (*OldName: newPV; Cycle: 5*)
	xFILTER_R_O2_NOxS_EngOut_A : FILTER_R := (0); (*FuB*) (*OldName: newPV; Cycle: 5*)
	xFILTER_R_O2_NOxS_EngOut_Avg : FILTER_R := (0); (*FuB*) (*OldName: newPV; Cycle: 5*)
	xFILTER_R_O2_NOxS_EngOut_B : FILTER_R := (0); (*FuB*) (*OldName: newPV; Cycle: 5*)
	xTOF_StartSpd_300s : TOF := (0); (*FuB*) (*OldName: newPV; Cycle: 5*)
	xTOF_StartSpd_900s : TOF := (0); (*FuB*) (*OldName: newPV; Cycle: 5*)
	xTON_CANwrite : TON := (0); (*FuB*) (*OldName: newPV; Cycle: 5*)
	xTON_DewP_CatOut : TON := (0); (*FuB*) (*OldName: newPV; Cycle: 5*)
	xTON_DewP_EngOut : TON := (0); (*FuB*) (*OldName: newPV; Cycle: 5*)
	xTON_GCB_On_60s : TON := (0); (*FuB*) (*OldName: newPV; Cycle: 5*)
	xTON_StdNOxS_CatOut_CAN_Ok : TON := (0); (*FuB*) (*OldName: newPV; Cycle: 5*)
	xTON_NOxS_CatOut_DiagDone : TON := (0); (*FuB*) (*OldName: newPV; Cycle: 5*)
	xTON_NOxS_EngOut_A_CAN_Ok : TON := (0); (*FuB*) (*OldName: newPV; Cycle: 5*)
	xTON_NOxS_EngOut_A_DiagDone : TON := (0); (*FuB*) (*OldName: newPV; Cycle: 5*)
	xTON_NOxS_EngOut_B_CAN_Ok : TON := (0); (*FuB*) (*OldName: newPV; Cycle: 5*)
	xTON_NOxS_EngOut_B_DiagDone : TON := (0); (*FuB*) (*OldName: newPV; Cycle: 5*)
	xTON_NOxS_EngOut_CAN_Ok : TON := (0); (*FuB*) (*OldName: newPV; Cycle: 5*)
	xTON_NOxS_EngOut_DiagDone : TON := (0); (*FuB*) (*OldName: newPV; Cycle: 5*)
	xTON_NOx_NOxS_EngOut_Dev_Hi : TON := (0); (*FuB*) (*OldName: newPV; Cycle: 5*)
	xTON_O2_NOxS_EngOut_Dev_Hi : TON := (0); (*FuB*) (*OldName: newPV; Cycle: 5*)
	xTON_RelMon_NOxS_EngOut : TON := (0); (*FuB*) (*OldName: newPV; Cycle: 5*)
	xTON_RelMon_NOxS_EngOut_A : TON := (0); (*FuB*) (*OldName: newPV; Cycle: 5*)
	xTON_RelMon_NOxS_EngOut_B : TON := (0); (*FuB*) (*OldName: newPV; Cycle: 5*)
	xTON_RelMon_NOx_NOxS_CatOut : TON := (0); (*FuB*) (*OldName: newPV; Cycle: 5*)
	xTON_RelMon_NOx_NOxS_EngOut : TON := (0); (*FuB*) (*OldName: newPV; Cycle: 5*)
	xTON_RelMon_NOx_NOxS_EngOut_A : TON := (0); (*FuB*) (*OldName: newPV; Cycle: 5*)
	xTON_RelMon_NOx_NOxS_EngOut_B : TON := (0); (*FuB*) (*OldName: newPV; Cycle: 5*)
	xTON_RelMon_O2_NOxS_CatOut : TON := (0); (*FuB*) (*OldName: newPV; Cycle: 5*)
	xTON_RelMon_O2_NOxS_EngOut : TON := (0); (*FuB*) (*OldName: newPV; Cycle: 5*)
	xTON_RelMon_O2_NOxS_EngOut_A : TON := (0); (*FuB*) (*OldName: newPV; Cycle: 5*)
	xTON_RelMon_O2_NOxS_EngOut_B : TON := (0); (*FuB*) (*OldName: newPV; Cycle: 5*)
	xTON_StartSpd_300s : TON := (0); (*FuB*) (*OldName: newPV; Cycle: 5*)
	xTON_StartSpd_600s : TON := (0); (*FuB*) (*OldName: newPV; Cycle: 5*)
	xTON_T_EG_Avg450_2m : TON := (0); (*FuB*) (*OldName: newPV; Cycle: 5*)
	xTON_LowNOxS_CatOut_CAN_Ok : TON; (*NOx sensor at CatOut low - Timer CAN is OK*) (*OldName: newPV; Cycle: 5*)
	xTON_LowNOxS_CatOut_CANcomm : TON := (0); (*NOx sensor at CatOut low - Timer CAN messages available*) (*OldName: newPV; Cycle: 5*)
	xTON_RelMon_NOxS_CatOut : TON := (0); (*NOx sensor at CatOut low - Timer release monitoring*) (*OldName: newPV; Cycle: 5*)
	xTON_Req_LowNOxS_CatOut_ID : TON := (0); (*NOx sensor at CatOut low - Timer request ID from module*) (*OldName: newPV; Cycle: 5*)
	bTON_LowNOxS_CatOut_CANErr : BOOL := 0; (*NOx sensor at CatOut low - Timer set variable - CAN communication error*) (*OldName: newPV; Cycle: 5*)
	rNOx_LowNOxS_CatOut : REAL := 0.0; (*NOx sensor at CatOut low - NOx wet value average from all queue messages [ppm]*) (*OldName: newPV; Cycle: 5*)
	rO2_LowNOxS_CatOut : REAL := 0.0; (*NOx sensor at CatOut low - O2 wet value average from all queue messages [%]*) (*OldName: newPV; Cycle: 5*)
	rk_NO2_LowNOxS_CatOut : REAL := 0; (*NOx sensor at CatOut low - Correction factor [%]*) (*OldName: newPV; Cycle: 5*)
	iLowNOxS_CatOut_ECM_ErrCode : INT := 0; (*NOx sensor at CatOut low - ECM error code received from module*) (*OldName: newPV; Cycle: 5*)
	bLowNOxS_CatOut_WarmUp : BOOL := 0; (*NOx sensor at CatOut low - Sensor is warming up*) (*OldName: newPV; Cycle: 5*)
	bLowNOxS_CatOut_SensorOff : BOOL := 0; (*NOx sensor at CatOut low - Sensor power is OFF*) (*OldName: newPV; Cycle: 5*)
	bLowNOxS_CatOut_BootUp : BOOL := 0; (*NOx sensor at CatOut low - Sensor is booting up*) (*OldName: newPV; Cycle: 5*)
	rCntO2_NOx_NOxS_CatOut_Ok : REAL := 0.0; (*NOx sensor at CatOut low - Counter of reliable messages read from queue*) (*OldName: newPV; Cycle: 5*)
	iCANwrite_LowNOxS_CatOut : ARRAY[0..7] OF USINT := [8(0)]; (*NOx sensor at CatOut low - CAN data to write in module*) (*OldName: newPV; Cycle: 5*)
	iCANwrite_LowNOxS_CatOut_ID : ARRAY[0..7] OF USINT := [8(0)]; (*NOx sensor at CatOut low - CAN data to request ID from module*) (*OldName: newPV; Cycle: 5*)
	iRead_LowNOxS_CatOut : ARRAY[0..7] OF USINT := [8(0)]; (*NOx sensor at CatOut low - CAN data read from module*) (*OldName: newPV; Cycle: 5*)
	iRead_LowNOxS_CatOut_Err : ARRAY[0..7] OF USINT := [8(0)]; (*NOx sensor at CatOut low - CAN data error message*) (*OldName: newPV; Cycle: 5*)
	iRead_LowNOxS_CatOut_HB : ARRAY[0..7] OF USINT := [8(0)]; (*NOx sensor at CatOut low - CAN data heartbeat message*) (*OldName: newPV; Cycle: 5*)
	iRead_LowNOxS_CatOut_ID : ARRAY[0..7] OF USINT := [8(0)]; (*NOx sensor at CatOut low - CAN data ID requested message*)
	xCANrd_LowNOxS_CatOut : CANrd := (0); (*NOx sensor at CatOut low - CAN queue read FBK*) (*OldName: newPV; Cycle: 5*)
	xCANwrite_LowNOxS_CatOut : CANwrite := (0); (*NOx sensor at CatOut low - CAN write FBK*) (*OldName: newPV; Cycle: 5*)
	xCANread_LowNOxS_CatOut_Err : CANread := (0); (*NOx sensor at CatOut low - CAN read FBK error message*) (*OldName: newPV; Cycle: 5*)
	xCANread_LowNOxS_CatOut : CANread := (0); (*NOx sensor at CatOut low - CAN read FBK requested ID message*) (*OldName: newPV; Cycle: 5*)
	xCANread_LowNOxS_CatOut_HB : CANread := (0); (*NOx sensor at CatOut low - CAN read FBK heartbeat message*) (*OldName: newPV; Cycle: 5*)
	bAMM_LowNOxS_CatOut_CANErr : BOOL := 0; (*NOx sensor CatOut low - CAN error from error message or reading*) (*OldName: newPV; Cycle: 5*)
	bAMM_LowNOxS_CANrd_CatOut : BOOL := 0; (*NOx sensor CatOut low - CAN failure reading queue*) (*OldName: newPV; Cycle: 5*)
	bAMM_LowNOxS_CatOut_Err : BOOL := 0; (*NOx sensor CatOut low - Error received from module*) (*OldName: newPV; Cycle: 5*)
	bQueue_NOxS2_IF3_Done : BOOL := 0; (*NOx sensor interface 3 queue open done*) (*OldName: newPV; Cycle: 5*)
	bReq_NOxS2_IF3_OpH	: BOOL := 0; (*request operating hours for Low NOx sensor (interface3)*) (*OldName: newPV; Cycle: 5*)
	bLowNOxS_CatOut_CAN_Ok : BOOL := 0; (*NOx sensor at CatOut low - CAN error read from module*) (*OldName: newPV; Cycle: 5*)
	iSt_LowNOxS_CatOut_Req : USINT := 0; (*NOx sensor at CatOut low - State machine to request IDs from module*) (*OldName: newPV; Cycle: 5*)
	bReq_NOxS2_IF3_ID : BOOL := 0; (*NOx sensor at CatOut low - Request ID form module*) (*OldName: newPV; Cycle: 5*)
	iID_LowNOxS_CatOut : ARRAY[0..3] OF UDINT := [4(0)]; (*NOx sensor at CatOut low - CAN identifiers for ID request*) (*OldName: newPV; Cycle: 5*)
	iRead_LowNOxS_CatOut_OpH : ARRAY[0..7] OF USINT := [8(0)]; (*CAN data read from module*) (*OldName: newPV; Cycle: 5*)
	iCANwrite_LowNOxS_CatOut_OpH : ARRAY[0..7] OF USINT := [8(0)]; (*CAN data sent to module*) (*OldName: newPV; Cycle: 5*)
	xCANwrite_LowNOxS_CatOut_OpH : CANwrite := (0); (*CAN write function*) (*OldName: newPV; Cycle: 5*)
	xCANread_LowNOxS_CatOut_OpH : CANread := (0); (*CAN read function*) (*OldName: newPV; Cycle: 5*)
	xTON_Req_LowNOxS_CatOut_OpH : TON := (0); (*Timer to read operating hours from low sensor module*) (*OldName: newPV; Cycle: 5*)
	bSTART_CntOpHours : BOOL := 0; (*Enable counting internal time on module*) (*OldName: newPV; Cycle: 5*)
	rOpHours_LowNOxS_CatOut : REAL := 0.0; (*Operating hours read from module - conversion [h]*) (*OldName: newPV; Cycle: 5*)
	iCnt_OpHours_LowNOxS_CatOut : UDINT := 0; (*NOx sensor at CatOut low - Operating hours read from module*) (*OldName: newPV; Cycle: 5*)
END_VAR
```

### Program Logical/Emission/SCR_Cat (IEC) - + SCR catalysator

- SCR_CatCyclic.st (not readable text: treated as protected, skipped)

#### SCR_Cat.var - Local variables
```iecst
VAR
	bErr_StopDosing : BOOL := FALSE; (*SCR General Error Flag --> Stop dosing --> Indicator Light ON*) (*V04.05.00.00*)
	bOnceShifting_2 : BOOL := FALSE; (*shifting only once*)
	bRelMon_AMM_2766 : BOOL := FALSE; (*release monitoring - at least one CAT temperature available*)
	bRelMon_Flow_UreaDosingOut : BOOL := FALSE; (*release monitoring - flow after urea dosing unit*)
	bRelMon_NO2_EMLine2 : BOOL := FALSE; (*release monitoring - NO2 in emission measurement line 2*)
	bRelMon_NO_EMLine2 : BOOL := FALSE; (*release monitoring - NO in emission measurement line 2*)
	bRelMon_O2_EMLine1 : BOOL := FALSE; (*release monitoring - O2 in emission measurement line 1*)
	bRelMon_Pr_CatIn : BOOL := FALSE; (*release monitoring - pressure before catalyst*)
	bRelMon_Pr_CatOut : BOOL := FALSE; (*release monitoring - pressure after catalyst*)
	bRelMon_Pr_ComprAirSupply : BOOL := FALSE; (*release monitoring - compressed air supply pressure *)
	bRelMon_Pr_UreaDosingIn : BOOL := FALSE; (*release monitoring - pressure before urea dosing unit*)
	bRelMon_Pr_UreaDosingOut : BOOL := FALSE; (*release monitoring - pressure after urea dosing unit*)
	bSCR_InjectValve_Open_Dem_Old : BOOL := FALSE; (*Save actual demand for Urea/Air injection valve - urea*)
	bSCR_InjectValve_Urea_Dem_Old : BOOL := FALSE; (*Save actual demand for Urea/Air injection valve - open*)
	bSCR_UreaDosingUnit2_Active_Old : BOOL := FALSE; (*Save actual used dosing unit*)
	i : INT := 0; (*auxiliary variable*)
	iCnt_AdjustCEMS_CO_1h : UINT := 0; (*counter - 1 hour average*)
	iCnt_AdjustCEMS_CO_5m : UINT := 0; (*counter - 5 min steady state*)
	iCnt_AdjustCEMS_NOxS_1h : UINT := 0; (*counter - 1 hour average*)
	iCnt_AdjustCEMS_NOxS_5m : UINT := 0; (*counter - 5 min steady state*)
	iCnt_AdjustCEMS_NOx_1h : UINT := 0; (*counter - 1 hour average*)
	iCnt_AdjustCEMS_NOx_5m : UINT := 0; (*counter - 5 min steady state*)
	iCnt_AirCompressor : UINT := 0; (*counter - Air compressor - seconds of operation *)
	iCnt_NH3SlipDetection : UINT := 0; (*counter - NH3 slip detection per hour*)
	iCnt_UreaDosingUnit : UINT := 0; (*counter - Urea dosing unit - seconds of operation *)
	iCnt_UreaDosingUnit2 : UINT := 0; (*counter - Urea dosing unit redundant - seconds of operation *)
	iSt_EM1_Purge : USINT := 0; (*State purging - emission measurement line1*)
	iSt_EM2_Purge : USINT := 0; (*State purging - emission measurement line2*)
	rCO_SCR_EMLine1_cor : REAL := 0; (*SCR Emission measurement line 1 - Offset corrected CO value [ppm]*)
	rCO_SCR_EMLine1_offset : REAL := 0; (*SCR Emission measurement line 1 - CO - Offset from external CEMS [ppm]*)
	rCO_SCR_EMLine1_Save : REAL := 0; (*SCR Emission measurement line 1 - Saved CO average value [ppm]*)
	rCO_SCR_EMLine1_valid : REAL := 0; (*SCR Emission measurement line 1 - Valid and 0-point corrected CO value [ppm]*)
	rNO2_SCR_EMLine1_cor : REAL := 0; (*SCR Emission measurement line 1 - 0-point corrected NO2 value [ppm]*)
	rNO2_SCR_EMLine1_Save : REAL := 0; (*SCR Emission measurement line 1 - Saved NO2 average value [ppm]*)
	rNO2_SCR_EMLine1_valid : REAL := 0; (*SCR Emission measurement line 1 - Valid and 0-point corrected NO2 value [ppm]*)
	rNO2_SCR_EMLine2_cor : REAL := 0; (*SCR Emission measurement line 2 - 0-point corrected NO2 value [ppm]*)
	rNO2_SCR_EMLine2_Save : REAL := 0; (*SCR Emission measurement line 2 - Saved NO2 average value [ppm]*)
	rNOx_NOxS_CatOut_offset : REAL := 0; (*SCR NOx sensor at catalyst outlet - Offset from external CEMS [ppm]*)
	rNOx_SCR_EMLine1_offset : REAL := 0; (*SCR Emission measurement line 1 - NOx - Offset from external CEMS [ppm]*)
	rNO_SCR_EMLine1_cor : REAL := 0; (*SCR Emission measurement line 1 - 0-point corrected NO value [ppm]*)
	rNO_SCR_EMLine1_Save : REAL := 0; (*SCR Emission measurement line 1 - Saved NO average value [ppm]*)
	rNO_SCR_EMLine1_valid : REAL := 0; (*SCR Emission measurement line 1 - Valid and 0-point corrected NO value [ppm]*)
	rNO_SCR_EMLine2_cor : REAL := 0; (*SCR Emission measurement line 2 - Offset corrected NO value [ppm]*)
	rNO_SCR_EMLine2_Save : REAL := 0; (*SCR Emission measurement line 2 - Saved NO average value [ppm]*)
	rTi_Lev_SCR_UreaTank_Lo : REAL := 0; (*Timer for tank level low - stop urea dosing*)
	xGR_MAXR_FlowUreaDosUnit : GR_MAXR := (0); (*FuB*)
	xGR_MAXR_P_Act_20 : GR_MAXR := (0); (*FuB*)
	xGR_MAXR_P_Act_Norm : GR_MAXR := (0); (*FuB*)
	xGR_MAXR_T_Rel_UreaSupplyPump : GR_MAXR := (0); (*FuB*)
	xGR_MAXR_T_SCR_Cat : GR_MAXR := (0); (*FuB*)
	xLCRMovAvgFlt_CO_5m : LCRMovAvgFlt := (0); (*FuB*)
	xLCRMovAvgFlt_CO_60m : LCRMovAvgFlt := (0); (*FuB*)
	xLCRMovAvgFlt_CO_Ext_5m : LCRMovAvgFlt := (0); (*FuB*)
	xLCRMovAvgFlt_CO_Ext_60m : LCRMovAvgFlt := (0); (*FuB*)
	xLCRMovAvgFlt_EMLine1_CO_5m : LCRMovAvgFlt := (0); (*FuB*)
	xLCRMovAvgFlt_EMLine1_CO_5s : LCRMovAvgFlt := (0); (*FuB*)
	xLCRMovAvgFlt_EMLine1_NO2_5m : LCRMovAvgFlt := (0); (*FuB*)
	xLCRMovAvgFlt_EMLine1_NO2_5s : LCRMovAvgFlt := (0); (*FuB*)
	xLCRMovAvgFlt_EMLine1_NO_5m : LCRMovAvgFlt := (0); (*FuB*)
	xLCRMovAvgFlt_EMLine1_NO_5s : LCRMovAvgFlt := (0); (*FuB*)
	xLCRMovAvgFlt_EMLine2_NO2_5m : LCRMovAvgFlt := (0); (*FuB*)
	xLCRMovAvgFlt_EMLine2_NO2_5s : LCRMovAvgFlt := (0); (*FuB*)
	xLCRMovAvgFlt_EMLine2_NO_5m : LCRMovAvgFlt := (0); (*FuB*)
	xLCRMovAvgFlt_EMLine2_NO_5s : LCRMovAvgFlt := (0); (*FuB*)
	xLCRMovAvgFlt_FlowUreaDosUnit : LCRMovAvgFlt; (*FuB*)
	xLCRMovAvgFlt_NOxS_5m : LCRMovAvgFlt := (0); (*FuB*)
	xLCRMovAvgFlt_NOxS_60m : LCRMovAvgFlt := (0); (*FuB*)
	xLCRMovAvgFlt_NOxS_Ext_5m : LCRMovAvgFlt := (0); (*FuB*)
	xLCRMovAvgFlt_NOxS_Ext_60m : LCRMovAvgFlt := (0); (*FuB*)
	xLCRMovAvgFlt_NOx_5m : LCRMovAvgFlt := (0); (*FuB*)
	xLCRMovAvgFlt_NOx_60m : LCRMovAvgFlt := (0); (*FuB*)
	xLCRMovAvgFlt_NOx_Ext_5m : LCRMovAvgFlt := (0); (*FuB*)
	xLCRMovAvgFlt_NOx_Ext_60m : LCRMovAvgFlt := (0); (*FuB*)
	xR_TRIG_AMM_2451 : R_TRIG := (0); (*FuB*)
	xR_TRIG_AMM_2453 : R_TRIG := (0); (*FuB*)
	xR_TRIG_AMM_3456 : R_TRIG := (0); (*FuB*)
	xR_TRIG_AMM_9380 : R_TRIG := (0); (*FuB*)
	xR_TRIG_Pump2_NotRdy : R_TRIG := (0); (*FuB*)
	xR_TRIG_Pump_NotRdy : R_TRIG := (0); (*FuB*)
	xSigScal_R_UreaDosingUnit_spMan : xSigScal_R := (0); (*FuB*)
	xTOF_bRel_SCR_UDC_2s : TOF := (0); (*FuB*)
	xTOF_bSCR_CemsExtCatOut_Rdy : TOF := (0); (*FuB*)
	xTOF_DFlow_SCR_UreaDosing_Hi : TOF := (0); (*FuB*)
	xTOF_DosingLimReached : TOF := (0); (*FuB*)
	xTOF_EMValve1_SGbOxi_Dem : TOF := (0); (*FuB*)
	xTOF_Overtravel_ComprAir : TOF := (0); (*FuB*)
	xTOF_Overtravel_EMPump1 : TOF := (0); (*FuB*)
	xTOF_Overtravel_EMPump2 : TOF := (0); (*FuB*)
	xTOF_Overtravel_InjectValve : TOF := (0); (*FuB*)
	xTOF_Overtravel_UreaSupply : TOF := (0); (*FuB*)
	xTOF_UreaDosingPumpFC_Reset : TOF := (0); (*FuB*)
	xTON_2453 : TON := (0); (*FuB*)
	xTON_3453 : TON := (0); (*FuB*)
	xTON_bSCR_Man_30m : TON := (0); (*FuB*)
	xTON_DFlow_SCR_UreaDosing_Hi : TON := (0); (*FuB*)
	xTON_DosingLimReached : TON := (0); (*FuB*)
	xTON_EMLine1_MsRdy : TON := (0); (*FuB*)
	xTON_EMLine1_OffsRdy : TON := (0); (*FuB*)
	xTON_EMLine2_MsRdy : TON := (0); (*FuB*)
	xTON_EMLine2_OffsRdy : TON := (0); (*FuB*)
	xTON_Eng_Run_5m : TON := (0); (*FuB*)
	xTON_GasAnalys_Purge_1 : TON := (0); (*FuB*)
	xTON_GasAnalys_Purge_2 : TON := (0); (*FuB*)
	xTON_GasAnalys_Purge_Inter_1 : TON := (0); (*FuB*)
	xTON_GasAnalys_Purge_Inter_2 : TON := (0); (*FuB*)
	xTON_GasAnalys_Purge_Shift : TON := (0); (*FuB*)
	xTON_GasAnalys_Waiting_1 : TON := (0); (*FuB*)
	xTON_GasAnalys_Waiting_2 : TON := (0); (*FuB*)
	xTON_NH3SlipDetect1 : TON := (0); (*FuB*)
	xTON_NH3SlipDetect2 : TON := (0); (*FuB*)
	xTON_NO2_SCR_EMLine1_MsErr : TON := (0); (*FuB*)
	xTON_NO2_SCR_EMLine2_MsErr : TON := (0); (*FuB*)
	xTON_NO_SCR_EMLine1_MsErr : TON := (0); (*FuB*)
	xTON_NO_SCR_EMLine2_MsErr : TON := (0); (*FuB*)
	xTON_Pr_UreaDosingOut_Hi : TON := (0); (*FuB*)
	xTON_P_Act_20 : TON := (0); (*FuB*)
	xTON_SecondTick : TON := (0); (*FuB*)
	xTON_T_SCR_Cat1 : TON := (0); (*FuB*)
	xTON_T_SCR_Cat2 : TON := (0); (*FuB*)
	xTON_UreaDosingPump2_NotRdy : TON := (0); (*FuB*)
	xTON_UreaDosingPump_NotRdy : TON := (0); (*FuB*)
	xTON_Urea_Err : TON := (0); (*FuB*)
	xTP_NH3SlipDetectComplete : TP; (*FuB*)
	xTP_NH3SlipDetectInterrupt : TP; (*FuB*)
	iTime_Meas : UDINT := 0;
	bTime_30sec : BOOL := 0;
	iTestTime : UDINT := 30000;
END_VAR
```

### Program Logical/Emission/SCR_UDC (IEC) - + SCR urea dosage controller

- SCR_UDCCyclic.st (not readable text: treated as protected, skipped)

- SCR_UDCInit.st (not readable text: treated as protected, skipped)

#### SCR_UDC.var - Local variables
```iecst
VAR
	bNOx_SCR_CatOut_Ok : BOOL := FALSE; (*NOx value after catalyst is ok and ready to use*)
	rCF_UreaFlow_H2 : REAL; (*Urea flow correction factor based on hydrogen*)
	rNOx_SCR_CatOut_act : REAL := 0; (*Actual NOx value after catalyst [ppm]*)
	xRamp_NOx_H2 : RAMPE_R; (*FuB*)
	xSigScal_NOx_H2 : xSigScal_R; (*Scaling of EngOut NOx setpoint based on H2*)
	xSigScal_NOx_P : xSigScal_R; (*Scaling of EngOut NOx setpoint based on power*)
	xTON_UreaFillUp : TON := (0); (*FuB*)
END_VAR
```

### Program Logical/Emission/SCR_MBSlave (IEC) - Modbus RTU Master IN/OUT data register

#### SCR_MBSlaveCyclic.st - Cyclic code
```iecst
(********************************************************************************************************************************************
SCR_MBSlave			 IN/OUT data register Modbus

This code is confidential and proprietary to the INNIO Company.
It may not be used in any form, or reproduced in any manner,
without written permission of the INNIO Company.
Copyright, INNIO Company, 2023

Customized modifications: -
------------------------

History:
-------
V04.04.00.00	02.08.2016	Pfanzagl		new
V04.04.01.00	02.06.2017	Denk			Adapted FOR SCR Modbus RTU Master
V04.05.00.00	28.07.2017	Tinello			Cleanup and connect of SCR variables
V04.09.00.00	27.11.2019	Tinello			Workaround if "urea/air injection valve - urea opened" - feedback is not available
V04.11.00.00	11.01.2022	Tinello			Bugfix: avoid negative urea flow rate signal
V04.13.00.00	21.11.2023	Tinello			Bugfix: Good quality only if para exist

*********************************************************************************************************************************************)
PROGRAM _CYCLIC

	(* Watchdog / generate ALIVE signal *)
	xTON_AliveBit_1(IN := NOT xTON_AliveBit_2.Q, PT := T#1s);
	xTON_AliveBit_2(IN :=     xTON_AliveBit_1.Q, PT := T#1s);

	(* ------------------------------------------------------------------------------------------------------------------------------------	*)
	(* ##################################################    OutData Register   ###########################################################	*)
	(* ------------------------------------------------------------------------------------------------------------------------------------	*)

	(* Register 1 *)
	OUT_EM.iModbus_SCR[1].0		:= OUT_EM.tSCR_ComprAirValve_Dem.Do;												(* air supply on *)
	OUT_EM.iModbus_SCR[1].1 	:= xTON_AliveBit_1.Q;																(* Alive *)
	OUT_EM.iModbus_SCR[1].2		:= 	   OUT_EM.tSCR_InjectValve_Urea_Dem.Do;											(* 3/2 - inject *)
	OUT_EM.iModbus_SCR[1].3		:= NOT OUT_EM.tSCR_InjectValve_Urea_Dem.Do;											(* 3/2 - purge *)
	OUT_EM.iModbus_SCR[1].4		:= bRel_Dosing OR (OUT_EM.tSCR_InjectValve_Urea_Dem.Do AND VIS2MM.bSCR_Man);		(* Injection enable	*)
	OUT_EM.iModbus_SCR[1].5		:= FALSE;																			(* Spare1_05 *)
	OUT_EM.iModbus_SCR[1].6		:= FALSE;																			(* Spare1_06 *)
	OUT_EM.iModbus_SCR[1].7		:= FALSE;																			(* Spare1_07 *)
	OUT_EM.iModbus_SCR[1].8		:= FALSE;																			(* Spare1_08 *)
	OUT_EM.iModbus_SCR[1].9		:= FALSE;																			(* Spare1_09 *)
	OUT_EM.iModbus_SCR[1].10	:= FALSE;																			(* Spare1_10 *)
	OUT_EM.iModbus_SCR[1].11	:= FALSE;																			(* Spare1_11 *)
	OUT_EM.iModbus_SCR[1].12	:= FALSE;																			(* Spare1_12 *)
	OUT_EM.iModbus_SCR[1].13	:= FALSE;																			(* Spare1_13 *)
	OUT_EM.iModbus_SCR[1].14	:= FALSE;																			(* Spare1_14 *)
	OUT_EM.iModbus_SCR[1].15	:= FALSE;																			(* Spare1_15 *)

	(* Register 2 - 10 *)
	OUT_EM.iModbus_SCR[2]		:= 0;    																			(* Spare_2 *)
	OUT_EM.iModbus_SCR[3]		:= REAL_TO_UINT(LIMIT(0, VIS2MM.rFlow_SCR_UreaDosingUnit_spMan 	* 100, 				(* Setpoint *)
														   Para.rFlow_SCR_UreaDosingUnit_Hi 	* 100 ));
	OUT_EM.iModbus_SCR[4]		:= REAL_TO_UINT(  		   Para.rFlow_SCR_UreaDosingUnit_Hi 	* 100);				(* Max. Flowrate *)
	OUT_EM.iModbus_SCR[5]		:= REAL_TO_UINT(Para.rPc_SCR_UreaSolution * 1000);									(* Urea water solultion *)
	OUT_EM.iModbus_SCR[6]		:= 0;    																			(* Spare_6 *)
	OUT_EM.iModbus_SCR[7]		:= 0;    																			(* Spare_7 *)
	OUT_EM.iModbus_SCR[8]		:= 0;    																			(* Spare_8 *)
	OUT_EM.iModbus_SCR[9]		:= 0;    																			(* Spare_9 *)
	OUT_EM.iModbus_SCR[10]		:= 0;   																			(* Spare_10 *)

	(* ------------------------------------------------------------------------------------------------------------------------------------	*)
	(* ##################################################    InData Register   ############################################################	*)
	(* ------------------------------------------------------------------------------------------------------------------------------------	*)
	MM2VIS.bSCR_SDB_Err[0] 			:= NOT IN_EM.iModbus_SCR_UINT[65].0;					(* On *)

		(* Check ALIVE signal *)
		xTON_AliveCheck_0(IN		:= NOT IN_EM.iModbus_SCR_UINT[65].1, PT:= T#5s);		(* Alive *)
		xTON_AliveCheck_1(IN		:= 	   IN_EM.iModbus_SCR_UINT[65].1, PT:= T#5s);

		bErr_SCR_BUS 				:= (xTON_AliveCheck_0.Q OR xTON_AliveCheck_1.Q) AND Para.bSCR_BUS_Exist;

	tInternSCR_InjectValve_Urea.Di 	:= 	   IN_EM.iModbus_SCR_UINT[65].2;					(* 3/2 - Position injection *)
	tInternSCR_InjectValve_Air.Di	:= 	   IN_EM.iModbus_SCR_UINT[65].3;					(* 3/2 - Position purging *)
	bConnectYourVariableHere 		:= 	   IN_EM.iModbus_SCR_UINT[65].4;					(* Door open *)
	OUT_EM.bSCR_SDB_EmStop 			:= NOT IN_EM.iModbus_SCR_UINT[65].5 AND		 			(* Emergency stop switch *)
										   Para.bSCR_BUS_Exist			AND
									   NOT (xTON_AliveCheck_0.Q OR xTON_AliveCheck_1.Q);
	bConnectYourVariableHere 		:= 	   IN_EM.iModbus_SCR_UINT[65].6;					(* Spare1_6 *)
	bConnectYourVariableHere 		:= 	   IN_EM.iModbus_SCR_UINT[65].7;					(* Spare1_7 *)
	bConnectYourVariableHere 		:= 	   IN_EM.iModbus_SCR_UINT[65].8;					(* Spare1_8 *)
	bConnectYourVariableHere 		:= 	   IN_EM.iModbus_SCR_UINT[65].9;					(* Spare1_9 *)
	bConnectYourVariableHere 		:= 	   IN_EM.iModbus_SCR_UINT[65].10;					(* Spare1_10 *)
	bConnectYourVariableHere 		:= 	   IN_EM.iModbus_SCR_UINT[65].11;					(* Spare1_11 *)
	bConnectYourVariableHere 		:=	   IN_EM.iModbus_SCR_UINT[65].12;					(* Spare1_12 *)
	bConnectYourVariableHere 		:= 	   IN_EM.iModbus_SCR_UINT[65].13;					(* Spare1_13 *)
	bConnectYourVariableHere 		:= 	   IN_EM.iModbus_SCR_UINT[65].14;					(* Spare1_14 *)
	bConnectYourVariableHere 		:= 	   IN_EM.iModbus_SCR_UINT[65].15;					(* Spare1_15 *)

	(*-------------------------------------------------------------------------------------------------------------------------------------	*)
	(* Register 66 *)
	iSCR_SDB_Status 				:= INT_TO_USINT(IN_EM.iModbus_SCR_UINT[66] / 256);		(* Status *)
	iConnectYourVariableHere1 		:= INT_TO_USINT(IN_EM.iModbus_SCR_UINT[66] MOD 256);	(* Spare66_1 *)

	(*-------------------------------------------------------------------------------------------------------------------------------------	*)
	(* Register 67 *)
	MM2VIS.bSCR_SDB_Err[1] 		:= IN_EM.iModbus_SCR_UINT[67].0;		(* Alarm 1:  Communication error to ECI *)
	MM2VIS.bSCR_SDB_Err[2] 		:= IN_EM.iModbus_SCR_UINT[67].1;		(* Alarm 2:  Emergency Stop active Smart Dosing Box *)
	MM2VIS.bSCR_SDB_Err[3] 		:= IN_EM.iModbus_SCR_UINT[67].2;		(* Alarm 3:  Hardware fault RS485 interface not connected *)
	MM2VIS.bSCR_SDB_Err[4] 		:= IN_EM.iModbus_SCR_UINT[67].3;		(* Alarm 4:  Hardware fault Analog input card not connected *)
	MM2VIS.bSCR_SDB_Err[5] 		:= IN_EM.iModbus_SCR_UINT[67].4;		(* Alarm 5:  Spare *)
	MM2VIS.bSCR_SDB_Err[6] 		:= IN_EM.iModbus_SCR_UINT[67].5;		(* Alarm 6:  DO Injection drive ON, short circuit or feedback voltage *)
	MM2VIS.bSCR_SDB_Err[7] 		:= IN_EM.iModbus_SCR_UINT[67].6;		(* Alarm 7:  DO air valve, short circuit or feedback voltage *)
	MM2VIS.bSCR_SDB_Err[8] 		:= IN_EM.iModbus_SCR_UINT[67].7;		(* Alarm 8:  DO Injection drive direction short circuit or feedb. volt.*)
	MM2VIS.bSCR_SDB_Err[9] 		:= IN_EM.iModbus_SCR_UINT[67].8;		(* Alarm 9:  DO Tact valve short circuit or feedback voltage *)
	MM2VIS.bSCR_SDB_Err[10] 	:= IN_EM.iModbus_SCR_UINT[67].9;		(* Alarm 10: Spare *)
	MM2VIS.bSCR_SDB_Err[11] 	:= IN_EM.iModbus_SCR_UINT[67].10;		(* Alarm 11: Analog Input 1: short circuit or out of range high *)
	MM2VIS.bSCR_SDB_Err[12] 	:= IN_EM.iModbus_SCR_UINT[67].11;		(* Alarm 12: Analog Input 1: cable break or out of range low *)
	MM2VIS.bSCR_SDB_Err[13] 	:= IN_EM.iModbus_SCR_UINT[67].12;		(* Alarm 13: Analog Input 2: short circuit or out of range high *)
	MM2VIS.bSCR_SDB_Err[14] 	:= IN_EM.iModbus_SCR_UINT[67].13;		(* Alarm 14: Analog Input 2: cable break or out of range low *)
	MM2VIS.bSCR_SDB_Err[15] 	:= IN_EM.iModbus_SCR_UINT[67].14;		(* Alarm 15: Analog Input 3: short circuit or out of range high *)
	MM2VIS.bSCR_SDB_Err[16] 	:= IN_EM.iModbus_SCR_UINT[67].15;		(* Alarm 16: Analog Input 3: cable break or out of range low *)

	(*-------------------------------------------------------------------------------------------------------------------------------------	*)
	(* Register 68 *)
	MM2VIS.bSCR_SDB_Err[17] 	:= IN_EM.iModbus_SCR_UINT[68].0;		(* Alarm 17: Spare *)
	MM2VIS.bSCR_SDB_Err[18] 	:= IN_EM.iModbus_SCR_UINT[68].1;		(* Alarm 18: Spare *)
	MM2VIS.bSCR_SDB_Err[19] 	:= IN_EM.iModbus_SCR_UINT[68].2;		(* Alarm 19: Spare *)
	MM2VIS.bSCR_SDB_Err[20] 	:= IN_EM.iModbus_SCR_UINT[68].3;		(* Alarm 20: Spare *)
	MM2VIS.bSCR_SDB_Err[21] 	:= IN_EM.iModbus_SCR_UINT[68].4;		(* Alarm 21: Spare *)
	MM2VIS.bSCR_SDB_Err[22] 	:= IN_EM.iModbus_SCR_UINT[68].5;		(* Alarm 22: Spare *)
	MM2VIS.bSCR_SDB_Err[23] 	:= IN_EM.iModbus_SCR_UINT[68].6;		(* Alarm 23: Spare *)
	MM2VIS.bSCR_SDB_Err[24] 	:= IN_EM.iModbus_SCR_UINT[68].7;		(* Alarm 24: Spare *)
	MM2VIS.bSCR_SDB_Err[25] 	:= IN_EM.iModbus_SCR_UINT[68].8;		(* Alarm 25: Internal CPU fault, memory fault, temperature fault *)
	MM2VIS.bSCR_SDB_Err[26] 	:= IN_EM.iModbus_SCR_UINT[68].9;		(* Warning 26: Spare *)
	MM2VIS.bSCR_SDB_Err[27] 	:= IN_EM.iModbus_SCR_UINT[68].10;		(* Warning 27: Spare *)
	MM2VIS.bSCR_SDB_Err[28] 	:= IN_EM.iModbus_SCR_UINT[68].11;		(* Warning 28: Reactant supply pressure to low *)
	MM2VIS.bSCR_SDB_Err[29] 	:= IN_EM.iModbus_SCR_UINT[68].12;		(* Warning 29: Reactant supply pressure to high *)
	MM2VIS.bSCR_SDB_Err[30] 	:= IN_EM.iModbus_SCR_UINT[68].13;		(* Warning 30: Spare *)
	MM2VIS.bSCR_SDB_Err[31] 	:= IN_EM.iModbus_SCR_UINT[68].14;		(* Warning 31: Actual flow dosing valve not ok *)
	MM2VIS.bSCR_SDB_Err[32] 	:= IN_EM.iModbus_SCR_UINT[68].15;		(* Warning 32: Actual position Injection valve "blow out" not valid *)

	(*-------------------------------------------------------------------------------------------------------------------------------------	*)
	(* Register 69 *)
	MM2VIS.bSCR_SDB_Err[33] 	:= IN_EM.iModbus_SCR_UINT[69].0;		(* Warning 33: Actual position Inection valve "Inject" not valid *)
	MM2VIS.bSCR_SDB_Err[34] 	:= IN_EM.iModbus_SCR_UINT[69].1;		(* Warning 34: Injection air pressure too low, cooling nozzel not ok *)
	MM2VIS.bSCR_SDB_Err[35] 	:= IN_EM.iModbus_SCR_UINT[69].2;		(* Warning 35: Injection air pressure too low for dosing *)
	MM2VIS.bSCR_SDB_Err[36] 	:= IN_EM.iModbus_SCR_UINT[69].3;		(* Warning 36: Injection air pressure too high *)
	MM2VIS.bSCR_SDB_Err[37] 	:= IN_EM.iModbus_SCR_UINT[69].4;		(* Warning 37: Spare *)
	MM2VIS.bSCR_SDB_Err[38] 	:= IN_EM.iModbus_SCR_UINT[69].5;		(* Warning 38: Spare *)
	MM2VIS.bSCR_SDB_Err[39] 	:= IN_EM.iModbus_SCR_UINT[69].6;		(* Warning 39: Spare *)
	MM2VIS.bSCR_SDB_Err[40] 	:= IN_EM.iModbus_SCR_UINT[69].7;		(* Warning 40: Spare *)
	MM2VIS.bSCR_SDB_Err[41] 	:= IN_EM.iModbus_SCR_UINT[69].8;		(* Warning 41: Spare *)
	MM2VIS.bSCR_SDB_Err[42] 	:= IN_EM.iModbus_SCR_UINT[69].9;		(* Warning 42: Spare *)
	MM2VIS.bSCR_SDB_Err[43] 	:= IN_EM.iModbus_SCR_UINT[69].10;		(* Warning 43: Spare *)
	MM2VIS.bSCR_SDB_Err[44] 	:= IN_EM.iModbus_SCR_UINT[69].11;		(* Warning 44: Spare *)
	MM2VIS.bSCR_SDB_Err[45] 	:= IN_EM.iModbus_SCR_UINT[69].12;		(* Warning 45: System not entirely purged or power loss dosing *)
	MM2VIS.bSCR_SDB_Err[46] 	:= IN_EM.iModbus_SCR_UINT[69].13;		(* Warning 46: Spare *)
	MM2VIS.bSCR_SDB_Err[47] 	:= IN_EM.iModbus_SCR_UINT[69].14;		(* Warning 47: Spare *)
	MM2VIS.bSCR_SDB_Err[48] 	:= IN_EM.iModbus_SCR_UINT[69].15;		(* Warning 48: Spare *)

	(*-------------------------------------------------------------------------------------------------------------------------------------	*)
	(* Register 70 - 84 *)
	iConnectYourVariableHere  				:= IN_EM.iModbus_SCR_UINT[70];						(* Spare70 *)

	tInternFlow_SCR_UreaDosingOut.Ai		:= UINT_TO_REAL(IN_EM.iModbus_SCR_UINT[71]) / 100;	(* Reactant - Flowrate *)
	tInternFlow_SCR_UreaDosingOut.Unfilt	:= UINT_TO_REAL(IN_EM.iModbus_SCR_UINT[71]) / 100;
	tInternFlow_SCR_UreaDosingOut.GoodQual	:= Para.bFlow_SCR_UreaDosingOut_Exist;

	iConnectYourVariableHere	  			:= IN_EM.iModbus_SCR_UINT[72];						(* Reactant - Max. Flowrate *)

	tInternPr_SCR_UreaDosingIn.Ai 			:= INT_TO_REAL(IN_EM.iModbus_SCR_INT[73]) / 1000;	(* Reactant - Feeding pressure *)
	tInternPr_SCR_UreaDosingIn.Unfilt 		:= INT_TO_REAL(IN_EM.iModbus_SCR_INT[73]) / 1000;
	tInternPr_SCR_UreaDosingIn.GoodQual		:= NOT MM2VIS.bSCR_SDB_Err[11] AND
											   NOT MM2VIS.bSCR_SDB_Err[12];

	tInternPr_SCR_UreaDosingOut.Ai 			:= INT_TO_REAL(IN_EM.iModbus_SCR_INT[74]) / 1000;	(* Reactant - Discharge pressure *)
	tInternPr_SCR_UreaDosingOut.Unfilt 		:= INT_TO_REAL(IN_EM.iModbus_SCR_INT[74]) / 1000;
	tInternPr_SCR_UreaDosingOut.GoodQual	:= NOT MM2VIS.bSCR_SDB_Err[13] AND
											   NOT MM2VIS.bSCR_SDB_Err[14];

	tInternPr_SCR_ComprAirSupply.Ai 		:= INT_TO_REAL(IN_EM.iModbus_SCR_INT[75]) / 1000;	(* Air - Pressure *)
	tInternPr_SCR_ComprAirSupply.Unfilt		:= INT_TO_REAL(IN_EM.iModbus_SCR_INT[75]) / 1000;
	tInternPr_SCR_ComprAirSupply.GoodQual	:= NOT MM2VIS.bSCR_SDB_Err[15] AND
										  	   NOT MM2VIS.bSCR_SDB_Err[16];

	iConnectYourVariableHere 				:= IN_EM.iModbus_SCR_UINT[76];						(* Spare12 *)
	iConnectYourVariableHere 				:= IN_EM.iModbus_SCR_UINT[77];						(* Spare13 *)
	iConnectYourVariableHere 				:= IN_EM.iModbus_SCR_UINT[78];						(* Spare14 *)
	iConnectYourVariableHere 				:= IN_EM.iModbus_SCR_UINT[79];						(* Spare15 *)
	iConnectYourVariableHere 				:= IN_EM.iModbus_SCR_UINT[80];						(* Spare16 *)
	iConnectYourVariableHere 				:= IN_EM.iModbus_SCR_UINT[81];						(* Spare17 *)
	iConnectYourVariableHere 				:= IN_EM.iModbus_SCR_UINT[82];						(* Spare18 *)
	iConnectYourVariableHere 				:= IN_EM.iModbus_SCR_UINT[83];						(* Spare19 *)
	iConnectYourVariableHere 				:= IN_EM.iModbus_SCR_UINT[84];						(* Spare20 *)

	(* ------------------------------------------------------------------------------------------------------------------------------------	*)
	(* ################################################   Inputs via Hardware   ###########################################################	*)
	(* ------------------------------------------------------------------------------------------------------------------------------------	*)
	IF NOT Para.bSCR_BUS_Exist THEN
		tInternSCR_InjectValve_Air			:= IN_EM.tSCR_InjectValve_Air;
		tInternFlow_SCR_UreaDosingOut		:= IN_EM.tFlow_SCR_UreaDosingOut;
		tInternPr_SCR_UreaDosingIn			:= IN_EM.tPr_SCR_UreaDosingIn;
		tInternPr_SCR_UreaDosingOut			:= IN_EM.tPr_SCR_UreaDosingOut;
		tInternPr_SCR_ComprAirSupply		:= IN_EM.tPr_SCR_ComprAirSupply;

		IF NOT IN_EM.tSCR_InjectValve_Urea.GoodQual THEN
			IF IN_EM.tSCR_InjectValve_Air.GoodQual
			THEN
				tInternSCR_InjectValve_Urea.Di 			:= NOT IN_EM.tSCR_InjectValve_Air.Di;
				tInternSCR_InjectValve_Urea.GoodQual	:=	   IN_EM.tSCR_InjectValve_Air.GoodQual;
			ELSE
				tInternSCR_InjectValve_Urea.Di 			:= FALSE;
				tInternSCR_InjectValve_Urea.GoodQual	:= FALSE;
			END_IF
		ELSE
			tInternSCR_InjectValve_Urea					:= IN_EM.tSCR_InjectValve_Urea;
		END_IF
	END_IF

	(* To avoid negative signal *)
	tInternFlow_SCR_UreaDosingOut.Ai		:= MAX(tInternFlow_SCR_UreaDosingOut.Ai, 	 0.001);
	tInternFlow_SCR_UreaDosingOut.Unfilt	:= MAX(tInternFlow_SCR_UreaDosingOut.Unfilt, 0.001);

END_PROGRAM
```

#### SCR_MBSlave.var - Local variables
```iecst
VAR
	bConnectYourVariableHere : BOOL := FALSE; (*Placeholder*)
	iConnectYourVariableHere : INT := 0; (*Placeholder*)
	iConnectYourVariableHere1 : USINT := 0; (*Placeholder*)
	iSCR_SDB_Status : USINT := 0; (*Status of SDB (smart dosing box) *)
	xTON_AliveBit_1 : TON := (0); (*Generate BUS ALIVE signal*)
	xTON_AliveBit_2 : TON := (0); (*Generate BUS ALIVE signal*)
	xTON_AliveCheck_0 : TON := (0); (*Check BUS ALIVE signal*)
	xTON_AliveCheck_1 : TON := (0); (*Check BUS ALIVE signal*)
END_VAR
```

### Program Logical/Emission/MsgEM (IEC) - Alarms generation
